LIN {X 0,Y 488.702,Z 333.231,A -85,B 0,C 180,E1 -6449.779,E2 -6449.779} C_VEL
LIN {X 0,Y 488.684,Z 333.228,A -85,B 0,C 180,E1 -6453.077,E2 -6453.077} C_VEL
LIN {X 0,Y 488.654,Z 333.238,A -85,B 0,C 180,E1 -6456.252,E2 -6456.252} C_VEL
LIN {X 0,Y 488.732,Z 333.224,A -85,B 0,C 180,E1 -6459.175,E2 -6459.175} C_VEL
LIN {X 0,Y 488.733,Z 333.22,A -85,B 0,C 180,E1 -6461.632,E2 -6461.632} C_VEL
LIN {X 0,Y 488.736,Z 333.23,A -85,B 0,C 180,E1 -6464.999,E2 -6464.999} C_VEL
LIN {X 0,Y 488.788,Z 333.224,A -85,B 0,C 180,E1 -6468.387,E2 -6468.387} C_VEL
LIN {X 0,Y 488.762,Z 333.222,A -85,B 0,C 180,E1 -6471.733,E2 -6471.733} C_VEL
LIN {X 0,Y 488.788,Z 333.223,A -85,B 0,C 180,E1 -6474.223,E2 -6474.223} C_VEL
LIN {X 0,Y 488.932,Z 333.202,A -85,B 0,C 180,E1 -6477.528,E2 -6477.528} C_VEL
LIN {X 0,Y 488.896,Z 333.211,A -85,B 0,C 180,E1 -6480.824,E2 -6480.824} C_VEL
LIN {X 0,Y 488.93,Z 333.21,A -85,B 0,C 180,E1 -6482.471,E2 -6482.471} C_VEL
LIN {X 0,Y 488.81,Z 333.217,A -85,B 0,C 180,E1 -6485.776,E2 -6485.776} C_VEL
LIN {X 0,Y 488.742,Z 333.23,A -85,B 0,C 180,E1 -6488.268,E2 -6488.268} C_VEL
LIN {X 0,Y 488.767,Z 333.222,A -85,B 0,C 180,E1 -6491.613,E2 -6491.613} C_VEL
LIN {X 0,Y 488.744,Z 333.227,A -85,B 0,C 180,E1 -6495.001,E2 -6495.001} C_VEL
LIN {X 0,Y 488.729,Z 333.235,A -85,B 0,C 180,E1 -6498.443,E2 -6498.443} C_VEL
LIN {X 0,Y 488.692,Z 333.227,A -85,B 0,C 180,E1 -6501.071,E2 -6501.071} C_VEL
LIN {X 0,Y 488.654,Z 333.233,A -85,B 0,C 180,E1 -6503.747,E2 -6503.747} C_VEL
LIN {X 0,Y 488.683,Z 333.233,A -85,B 0,C 180,E1 -6506.922,E2 -6506.922} C_VEL
LIN {X 0,Y 488.701,Z 333.232,A -85,B 0,C 180,E1 -6510.221,E2 -6510.221} C_VEL
LIN {X 0,Y 488.696,Z 333.23,A -85,B 0,C 180,E1 -6513.481,E2 -6513.481} C_VEL
LIN {X 0,Y 488.635,Z 333.246,A -85,B 0,C 180,E1 -6516.35,E2 -6516.35} C_VEL
LIN {X 0,Y 488.661,Z 333.236,A -85,B 0,C 180,E1 -6519.258,E2 -6519.258} C_VEL
LIN {X 0,Y 488.636,Z 333.244,A -85,B 0,C 180,E1 -6522.532,E2 -6522.532} C_VEL
LIN {X 0,Y 488.684,Z 333.234,A -85,B 0,C 180,E1 -6525.198,E2 -6525.198} C_VEL
LIN {X 0,Y 488.632,Z 333.245,A -85,B 0,C 180,E1 -6528.579,E2 -6528.579} C_VEL
LIN {X 0,Y 488.64,Z 333.243,A -85,B 0,C 180,E1 -6531.798,E2 -6531.798} C_VEL
LIN {X 0,Y 488.704,Z 333.232,A -85,B 0,C 180,E1 -6535.056,E2 -6535.056} C_VEL
LIN {X 0,Y 488.685,Z 333.24,A -85,B 0,C 180,E1 -6538.05,E2 -6538.05} C_VEL
LIN {X 0,Y 488.692,Z 333.232,A -85,B 0,C 180,E1 -6540.729,E2 -6540.729} C_VEL
LIN {X 0,Y 488.709,Z 333.391,A -85,B 0,C 180,E1 -6543.9,E2 -6543.9} C_VEL
LIN {X 0,Y 491.166,Z 344.956,A -85,B 0,C 180,E1 -6545.98,E2 -6545.98} C_VEL
LIN {X 0,Y 491.203,Z 350.07,A -85,B 0,C 180,E1 -6546.832,E2 -6546.832} C_VEL
LIN {X 0,Y 490.392,Z 368.886,A -85,B 0,C 180,E1 -6549.884,E2 -6549.884} C_VEL
LIN {X 0,Y 490.314,Z 371.302,A -85,B 0,C 180,E1 -6550.273,E2 -6550.273} C_VEL
LIN {X 0,Y 493.534,Z 389.01,A -85,B 0,C 180,E1 -6550.687,E2 -6550.687} C_VEL
LIN {X 0,Y 492.513,Z 509.403,A -85,B 0,C 180,E1 -6552.484,E2 -6552.484} C_VEL
LIN {X 0,Y 492.126,Z 523.948,A -85,B 0,C 180,E1 -6552.874,E2 -6552.874} C_VEL
LIN {X 0,Y 491.704,Z 538.324,A -85,B 0,C 180,E1 -6553.444,E2 -6553.444} C_VEL
LIN {X 0,Y 491.255,Z 551.142,A -85,B 0,C 180,E1 -6554.123,E2 -6554.123} C_VEL
LIN {X 0,Y 490.687,Z 563.612,A -85,B 0,C 180,E1 -6554.955,E2 -6554.955} C_VEL
LIN {X 0,Y 490.137,Z 575.001,A -85,B 0,C 180,E1 -6555.893,E2 -6555.893} C_VEL
LIN {X 0,Y 489.549,Z 585.47,A -85,B 0,C 180,E1 -6556.933,E2 -6556.933} C_VEL
LIN {X 0,Y 489.174,Z 596.158,A -85,B 0,C 180,E1 -6558.224,E2 -6558.224} C_VEL
LIN {X 0,Y 488.668,Z 605.74,A -85,B 0,C 180,E1 -6559.645,E2 -6559.645} C_VEL
LIN {X 0,Y 488.349,Z 613.708,A -85,B 0,C 180,E1 -6561.102,E2 -6561.102} C_VEL
LIN {X 0,Y 488.106,Z 620.121,A -85,B 0,C 180,E1 -6562.556,E2 -6562.556} C_VEL
LIN {X 0,Y 488.051,Z 625.81,A -85,B 0,C 180,E1 -6564.216,E2 -6564.216} C_VEL
LIN {X 0,Y 487.909,Z 629.938,A -85,B 0,C 180,E1 -6565.871,E2 -6565.871} C_VEL
LIN {X 0,Y 487.955,Z 631.458,A -85,B 0,C 180,E1 -6566.699,E2 -6566.699} C_VEL
LIN {X 0,Y 487.885,Z 633.463,A -85,B 0,C 180,E1 -6568.35,E2 -6568.35} C_VEL
LIN {X 0,Y 487.817,Z 634.126,A -85,B 0,C 180,E1 -6570.001,E2 -6570.001} C_VEL
LIN {X 0,Y 487.886,Z 633.459,A -85,B 0,C 180,E1 -6571.652,E2 -6571.652} C_VEL
LIN {X 0,Y 487.956,Z 631.449,A -85,B 0,C 180,E1 -6573.304,E2 -6573.304} C_VEL
LIN {X 0,Y 487.962,Z 628.05,A -85,B 0,C 180,E1 -6574.959,E2 -6574.959} C_VEL
LIN {X 0,Y 488.042,Z 623.66,A -85,B 0,C 180,E1 -6576.472,E2 -6576.472} C_VEL
LIN {X 0,Y 488.17,Z 618.444,A -85,B 0,C 180,E1 -6577.862,E2 -6577.862} C_VEL
LIN {X 0,Y 488.422,Z 611.598,A -85,B 0,C 180,E1 -6579.317,E2 -6579.317} C_VEL
LIN {X 0,Y 488.818,Z 603.102,A -85,B 0,C 180,E1 -6580.774,E2 -6580.774} C_VEL
LIN {X 0,Y 489.194,Z 594.847,A -85,B 0,C 180,E1 -6581.946,E2 -6581.946} C_VEL
LIN {X 0,Y 489.581,Z 585.447,A -85,B 0,C 180,E1 -6583.068,E2 -6583.068} C_VEL
LIN {X 0,Y 490.123,Z 574.974,A -85,B 0,C 180,E1 -6584.11,E2 -6584.11} C_VEL
LIN {X 0,Y 490.661,Z 563.574,A -85,B 0,C 180,E1 -6585.048,E2 -6585.048} C_VEL
LIN {X 0,Y 491.228,Z 551.097,A -85,B 0,C 180,E1 -6585.881,E2 -6585.881} C_VEL
LIN {X 0,Y 491.808,Z 537.148,A -85,B 0,C 180,E1 -6586.608,E2 -6586.608} C_VEL
LIN {X 0,Y 492.15,Z 523.043,A -85,B 0,C 180,E1 -6587.157,E2 -6587.157} C_VEL
LIN {X 0,Y 492.538,Z 509.287,A -85,B 0,C 180,E1 -6587.518,E2 -6587.518} C_VEL
LIN {X 0,Y 493.537,Z 388.937,A -85,B 0,C 180,E1 -6589.313,E2 -6589.313} C_VEL
LIN {X 0,Y 490.294,Z 371.281,A -85,B 0,C 180,E1 -6589.73,E2 -6589.73} C_VEL
LIN {X 0,Y 491.158,Z 351.392,A -85,B 0,C 180,E1 -6592.951,E2 -6592.951} C_VEL
LIN {X 0,Y 491.288,Z 346.01,A -85,B 0,C 180,E1 -6593.837,E2 -6593.837} C_VEL
LIN {X 0,Y 488.696,Z 333.239,A -85,B 0,C 180,E1 -6596.132,E2 -6596.132} C_VEL
LIN {X 0,Y 488.703,Z 333.237,A -85,B 0,C 180,E1 -6599.273,E2 -6599.273} C_VEL
LIN {X 0,Y 488.707,Z 333.233,A -85,B 0,C 180,E1 -6602.148,E2 -6602.148} C_VEL
LIN {X 0,Y 488.72,Z 333.234,A -85,B 0,C 180,E1 -6605.116,E2 -6605.116} C_VEL
LIN {X 0,Y 488.682,Z 333.234,A -85,B 0,C 180,E1 -6608.201,E2 -6608.201} C_VEL
LIN {X 0,Y 488.723,Z 333.229,A -85,B 0,C 180,E1 -6610.345,E2 -6610.345} C_VEL
LIN {X 0,Y 488.691,Z 333.234,A -85,B 0,C 180,E1 -6613.655,E2 -6613.655} C_VEL
LIN {X 0,Y 488.692,Z 333.237,A -85,B 0,C 180,E1 -6616.346,E2 -6616.346} C_VEL
LIN {X 0,Y 488.738,Z 333.228,A -85,B 0,C 180,E1 -6619.677,E2 -6619.677} C_VEL
LIN {X 0,Y 488.675,Z 333.238,A -85,B 0,C 180,E1 -6622.841,E2 -6622.841} C_VEL
LIN {X 0,Y 488.735,Z 333.231,A -85,B 0,C 180,E1 -6625.888,E2 -6625.888} C_VEL
LIN {X 0,Y 488.697,Z 333.236,A -85,B 0,C 180,E1 -6628.821,E2 -6628.821} C_VEL
LIN {X 0,Y 488.714,Z 333.239,A -85,B 0,C 180,E1 -6631.669,E2 -6631.669} C_VEL
LIN {X 0,Y 488.702,Z 333.235,A -85,B 0,C 180,E1 -6634.96,E2 -6634.96} C_VEL
LIN {X 0,Y 488.739,Z 333.298,A -85,B 0,C 180,E1 -6636.726,E2 -6636.726} C_VEL
LIN {X 0,Y 490.353,Z 342.584,A -85,B 0,C 180,E1 -6638.308,E2 -6638.308} C_VEL
LIN {X 0,Y 490.033,Z 361.132,A -85,B 0,C 180,E1 -6641.346,E2 -6641.346} C_VEL
LIN {X 0,Y 489.795,Z 376.155,A -85,B 0,C 180,E1 -6643.82,E2 -6643.82} C_VEL
LIN {X 0,Y 491.76,Z 387.528,A -85,B 0,C 180,E1 -6644.09,E2 -6644.09} C_VEL
LIN {X 0,Y 490.807,Z 484.773,A -85,B 0,C 180,E1 -6645.7,E2 -6645.7} C_VEL
LIN {X 0,Y 490.587,Z 497.505,A -85,B 0,C 180,E1 -6646.063,E2 -6646.063} C_VEL
LIN {X 0,Y 490.274,Z 509.826,A -85,B 0,C 180,E1 -6646.583,E2 -6646.583} C_VEL
LIN {X 0,Y 489.978,Z 521.787,A -85,B 0,C 180,E1 -6647.256,E2 -6647.256} C_VEL
LIN {X 0,Y 489.692,Z 533.257,A -85,B 0,C 180,E1 -6648.094,E2 -6648.094} C_VEL
LIN {X 0,Y 489.302,Z 543.523,A -85,B 0,C 180,E1 -6649.029,E2 -6649.029} C_VEL
LIN {X 0,Y 488.952,Z 552.812,A -85,B 0,C 180,E1 -6650.068,E2 -6650.068} C_VEL
LIN {X 0,Y 488.605,Z 561.725,A -85,B 0,C 180,E1 -6651.313,E2 -6651.313} C_VEL
LIN {X 0,Y 488.371,Z 568.89,A -85,B 0,C 180,E1 -6652.558,E2 -6652.558} C_VEL
LIN {X 0,Y 488.235,Z 575.028,A -85,B 0,C 180,E1 -6653.912,E2 -6653.912} C_VEL
LIN {X 0,Y 487.996,Z 579.059,A -85,B 0,C 180,E1 -6655.043,E2 -6655.043} C_VEL
LIN {X 0,Y 488.112,Z 581.377,A -85,B 0,C 180,E1 -6655.872,E2 -6655.872} C_VEL
LIN {X 0,Y 488.025,Z 583.275,A -85,B 0,C 180,E1 -6656.698,E2 -6656.698} C_VEL
LIN {X 0,Y 488,Z 584.743,A -85,B 0,C 180,E1 -6657.524,E2 -6657.524} C_VEL
LIN {X 0,Y 487.837,Z 586.379,A -85,B 0,C 180,E1 -6659.175,E2 -6659.175} C_VEL
LIN {X 0,Y 487.825,Z 586.609,A -85,B 0,C 180,E1 -6660,E2 -6660} C_VEL
LIN {X 0,Y 487.837,Z 586.402,A -85,B 0,C 180,E1 -6660.826,E2 -6660.826} C_VEL
LIN {X 0,Y 487.994,Z 584.776,A -85,B 0,C 180,E1 -6662.476,E2 -6662.476} C_VEL
LIN {X 0,Y 487.999,Z 583.356,A -85,B 0,C 180,E1 -6663.303,E2 -6663.303} C_VEL
LIN {X 0,Y 488.055,Z 580.39,A -85,B 0,C 180,E1 -6664.543,E2 -6664.543} C_VEL
LIN {X 0,Y 488.226,Z 575.193,A -85,B 0,C 180,E1 -6666.086,E2 -6666.086} C_VEL
LIN {X 0,Y 488.304,Z 569.158,A -85,B 0,C 180,E1 -6667.443,E2 -6667.443} C_VEL
LIN {X 0,Y 488.581,Z 562.093,A -85,B 0,C 180,E1 -6668.687,E2 -6668.687} C_VEL
LIN {X 0,Y 488.904,Z 553.302,A -85,B 0,C 180,E1 -6669.933,E2 -6669.933} C_VEL
LIN {X 0,Y 489.268,Z 544.258,A -85,B 0,C 180,E1 -6670.972,E2 -6670.972} C_VEL
LIN {X 0,Y 489.6,Z 534.233,A -85,B 0,C 180,E1 -6671.908,E2 -6671.908} C_VEL
LIN {X 0,Y 489.938,Z 522.917,A -85,B 0,C 180,E1 -6672.761,E2 -6672.761} C_VEL
LIN {X 0,Y 490.276,Z 510.773,A -85,B 0,C 180,E1 -6673.47,E2 -6673.47} C_VEL
LIN {X 0,Y 490.621,Z 497.552,A -85,B 0,C 180,E1 -6674.042,E2 -6674.042} C_VEL
LIN {X 0,Y 490.877,Z 485.355,A -85,B 0,C 180,E1 -6674.404,E2 -6674.404} C_VEL
LIN {X 0,Y 491.124,Z 459.02,A -85,B 0,C 180,E1 -6674.847,E2 -6674.847} C_VEL
LIN {X 0,Y 491.597,Z 386.183,A -85,B 0,C 180,E1 -6676.007,E2 -6676.007} C_VEL
LIN {X 0,Y 489.573,Z 374.944,A -85,B 0,C 180,E1 -6676.262,E2 -6676.262} C_VEL
LIN {X 0,Y 489.986,Z 357.352,A -85,B 0,C 180,E1 -6679.263,E2 -6679.263} C_VEL
LIN {X 0,Y 490.237,Z 342.024,A -85,B 0,C 180,E1 -6681.884,E2 -6681.884} C_VEL
LIN {X 0,Y 488.753,Z 333.23,A -85,B 0,C 180,E1 -6683.467,E2 -6683.467} C_VEL
LIN {X 0,Y 488.797,Z 333.221,A -85,B 0,C 180,E1 -6686.943,E2 -6686.943} C_VEL
LIN {X 0,Y 488.715,Z 333.233,A -85,B 0,C 180,E1 -6690.363,E2 -6690.363} C_VEL
LIN {X 0,Y 488.74,Z 333.228,A -85,B 0,C 180,E1 -6693.484,E2 -6693.484} C_VEL
LIN {X 0,Y 488.678,Z 333.238,A -85,B 0,C 180,E1 -6696.353,E2 -6696.353} C_VEL
LIN {X 0,Y 488.699,Z 333.232,A -85,B 0,C 180,E1 -6699.255,E2 -6699.255} C_VEL
LIN {X 0,Y 488.693,Z 333.233,A -85,B 0,C 180,E1 -6702.526,E2 -6702.526} C_VEL
LIN {X 0,Y 488.693,Z 333.234,A -85,B 0,C 180,E1 -6705.431,E2 -6705.431} C_VEL
LIN {X 0,Y 488.681,Z 333.234,A -85,B 0,C 180,E1 -6708.581,E2 -6708.581} C_VEL
LIN {X 0,Y 488.667,Z 333.236,A -85,B 0,C 180,E1 -6709.017,E2 -6709.017} C_VEL
LIN {X 0,Y 488.004,Z 333.325,A -85,B 0,C 180,E1 -6709.705,E2 -6709.705} C_VEL
LIN {X 0,Y 485.141,Z 333.677,A -85,B 0,C 180,E1 -6710.822,E2 -6710.822} C_VEL
LIN {X 0,Y 482.717,Z 333.983,A -85,B 0,C 180,E1 -6711.722,E2 -6711.722} C_VEL
LIN {X 0,Y 481.679,Z 334.108,A -85,B 0,C 180,E1 -6712.418,E2 -6712.418} C_VEL
LIN {X 0,Y 481.596,Z 334.118,A -85,B 0,C 180,E1 -6712.653,E2 -6712.653} C_VEL
LIN {X 0,Y 481.683,Z 334.11,A -85,B 0,C 180,E1 -6715.316,E2 -6715.316} C_VEL
LIN {X 0,Y 481.627,Z 334.115,A -85,B 0,C 180,E1 -6718.309,E2 -6718.309} C_VEL
LIN {X 0,Y 481.657,Z 334.117,A -85,B 0,C 180,E1 -6721.215,E2 -6721.215} C_VEL
LIN {X 0,Y 481.621,Z 334.119,A -85,B 0,C 180,E1 -6724.037,E2 -6724.037} C_VEL
LIN {X 0,Y 481.639,Z 334.155,A -85,B 0,C 180,E1 -6724.823,E2 -6724.823} C_VEL
LIN {X 0,Y 484.1,Z 346.337,A -85,B 0,C 180,E1 -6727.147,E2 -6727.147} C_VEL
LIN {X 0,Y 483.546,Z 360.333,A -85,B 0,C 180,E1 -6729.584,E2 -6729.584} C_VEL
LIN {X 0,Y 483.402,Z 362.996,A -85,B 0,C 180,E1 -6730.041,E2 -6730.041} C_VEL
LIN {X 0,Y 486.825,Z 379.799,A -85,B 0,C 180,E1 -6730.449,E2 -6730.449} C_VEL
LIN {X 0,Y 485.833,Z 498.193,A -85,B 0,C 180,E1 -6732.232,E2 -6732.232} C_VEL
LIN {X 0,Y 485.466,Z 512.773,A -85,B 0,C 180,E1 -6732.595,E2 -6732.595} C_VEL
LIN {X 0,Y 485.165,Z 526.114,A -85,B 0,C 180,E1 -6733.099,E2 -6733.099} C_VEL
LIN {X 0,Y 484.665,Z 537.87,A -85,B 0,C 180,E1 -6733.682,E2 -6733.682} C_VEL
LIN {X 0,Y 484.068,Z 551.218,A -85,B 0,C 180,E1 -6734.526,E2 -6734.526} C_VEL
LIN {X 0,Y 483.463,Z 563.197,A -85,B 0,C 180,E1 -6735.476,E2 -6735.476} C_VEL
LIN {X 0,Y 482.834,Z 574.12,A -85,B 0,C 180,E1 -6736.532,E2 -6736.532} C_VEL
LIN {X 0,Y 482.362,Z 584.598,A -85,B 0,C 180,E1 -6737.764,E2 -6737.764} C_VEL
LIN {X 0,Y 481.876,Z 593.784,A -85,B 0,C 180,E1 -6739.069,E2 -6739.069} C_VEL
LIN {X 0,Y 481.475,Z 602.295,A -85,B 0,C 180,E1 -6740.547,E2 -6740.547} C_VEL
LIN {X 0,Y 481.176,Z 609.155,A -85,B 0,C 180,E1 -6742.023,E2 -6742.023} C_VEL
LIN {X 0,Y 481.033,Z 614.484,A -85,B 0,C 180,E1 -6743.463,E2 -6743.463} C_VEL
LIN {X 0,Y 480.898,Z 618.792,A -85,B 0,C 180,E1 -6744.968,E2 -6744.968} C_VEL
LIN {X 0,Y 480.887,Z 622.208,A -85,B 0,C 180,E1 -6746.647,E2 -6746.647} C_VEL
LIN {X 0,Y 480.791,Z 624.243,A -85,B 0,C 180,E1 -6748.323,E2 -6748.323} C_VEL
LIN {X 0,Y 480.742,Z 624.947,A -85,B 0,C 180,E1 -6749.999,E2 -6749.999} C_VEL
LIN {X 0,Y 480.79,Z 624.327,A -85,B 0,C 180,E1 -6751.674,E2 -6751.674} C_VEL
LIN {X 0,Y 480.886,Z 622.372,A -85,B 0,C 180,E1 -6753.35,E2 -6753.35} C_VEL
LIN {X 0,Y 480.897,Z 619.029,A -85,B 0,C 180,E1 -6755.029,E2 -6755.029} C_VEL
LIN {X 0,Y 481.012,Z 614.202,A -85,B 0,C 180,E1 -6756.711,E2 -6756.711} C_VEL
LIN {X 0,Y 481.246,Z 607.745,A -85,B 0,C 180,E1 -6758.396,E2 -6758.396} C_VEL
LIN {X 0,Y 481.578,Z 600.556,A -85,B 0,C 180,E1 -6759.872,E2 -6759.872} C_VEL
LIN {X 0,Y 481.938,Z 593.021,A -85,B 0,C 180,E1 -6761.139,E2 -6761.139} C_VEL
LIN {X 0,Y 482.299,Z 584.534,A -85,B 0,C 180,E1 -6762.337,E2 -6762.337} C_VEL
LIN {X 0,Y 482.82,Z 574.963,A -85,B 0,C 180,E1 -6763.466,E2 -6763.466} C_VEL
LIN {X 0,Y 483.398,Z 564.21,A -85,B 0,C 180,E1 -6764.523,E2 -6764.523} C_VEL
LIN {X 0,Y 484.013,Z 552.449,A -85,B 0,C 180,E1 -6765.473,E2 -6765.473} C_VEL
LIN {X 0,Y 484.521,Z 541.228,A -85,B 0,C 180,E1 -6766.212,E2 -6766.212} C_VEL
LIN {X 0,Y 485.086,Z 528.046,A -85,B 0,C 180,E1 -6766.901,E2 -6766.901} C_VEL
LIN {X 0,Y 485.484,Z 513.858,A -85,B 0,C 180,E1 -6767.457,E2 -6767.457} C_VEL
LIN {X 0,Y 485.818,Z 500.184,A -85,B 0,C 180,E1 -6767.82,E2 -6767.82} C_VEL
LIN {X 0,Y 486.905,Z 380.439,A -85,B 0,C 180,E1 -6769.629,E2 -6769.629} C_VEL
LIN {X 0,Y 483.411,Z 362.985,A -85,B 0,C 180,E1 -6770.052,E2 -6770.052} C_VEL
LIN {X 0,Y 484.112,Z 346.87,A -85,B 0,C 180,E1 -6772.849,E2 -6772.849} C_VEL
LIN {X 0,Y 482.469,Z 337.99,A -85,B 0,C 180,E1 -6774.527,E2 -6774.527} C_VEL
LIN {X 0,Y 481.632,Z 334.12,A -85,B 0,C 180,E1 -6775.284,E2 -6775.284} C_VEL
LIN {X 0,Y 481.643,Z 334.115,A -85,B 0,C 180,E1 -6777.834,E2 -6777.834} C_VEL
LIN {X 0,Y 481.624,Z 334.121,A -85,B 0,C 180,E1 -6780.711,E2 -6780.711} C_VEL
LIN {X 0,Y 481.669,Z 334.111,A -85,B 0,C 180,E1 -6783.728,E2 -6783.728} C_VEL
LIN {X 0,Y 481.611,Z 334.121,A -85,B 0,C 180,E1 -6786.746,E2 -6786.746} C_VEL
LIN {X 0,Y 481.647,Z 334.11,A -85,B 0,C 180,E1 -6789.941,E2 -6789.941} C_VEL
LIN {X 0,Y 481.609,Z 334.118,A -85,B 0,C 180,E1 -6793.301,E2 -6793.301} C_VEL
LIN {X 0,Y 481.642,Z 334.111,A -85,B 0,C 180,E1 -6795.64,E2 -6795.64} C_VEL
LIN {X 0,Y 481.615,Z 334.121,A -85,B 0,C 180,E1 -6798.954,E2 -6798.954} C_VEL
LIN {X 0,Y 481.637,Z 334.106,A -85,B 0,C 180,E1 -6801.993,E2 -6801.993} C_VEL
LIN {X 0,Y 481.669,Z 334.108,A -85,B 0,C 180,E1 -6805.316,E2 -6805.316} C_VEL
LIN {X 0,Y 481.626,Z 334.109,A -85,B 0,C 180,E1 -6808.31,E2 -6808.31} C_VEL
LIN {X 0,Y 481.645,Z 334.111,A -85,B 0,C 180,E1 -6811.215,E2 -6811.215} C_VEL
LIN {X 0,Y 481.615,Z 334.105,A -85,B 0,C 180,E1 -6814.038,E2 -6814.038} C_VEL
LIN {X 0,Y 481.66,Z 334.115,A -85,B 0,C 180,E1 -6816.811,E2 -6816.811} C_VEL
LIN {X 0,Y 481.679,Z 334.1,A -85,B 0,C 180,E1 -6819.502,E2 -6819.502} C_VEL
LIN {X 0,Y 481.67,Z 334.101,A -85,B 0,C 180,E1 -6822.157,E2 -6822.157} C_VEL
LIN {X 0,Y 481.721,Z 334.107,A -85,B 0,C 180,E1 -6824.775,E2 -6824.775} C_VEL
LIN {X 0,Y 481.734,Z 334.101,A -85,B 0,C 180,E1 -6828.215,E2 -6828.215} C_VEL
LIN {X 0,Y 481.718,Z 334.099,A -85,B 0,C 180,E1 -6831.611,E2 -6831.611} C_VEL
LIN {X 0,Y 481.749,Z 334.099,A -85,B 0,C 180,E1 -6834.139,E2 -6834.139} C_VEL
LIN {X 0,Y 481.898,Z 334.078,A -85,B 0,C 180,E1 -6837.492,E2 -6837.492} C_VEL
LIN {X 0,Y 481.848,Z 334.089,A -85,B 0,C 180,E1 -6840.836,E2 -6840.836} C_VEL
LIN {X 0,Y 481.896,Z 334.087,A -85,B 0,C 180,E1 -6842.508,E2 -6842.508} C_VEL
LIN {X 0,Y 481.769,Z 334.095,A -85,B 0,C 180,E1 -6845.861,E2 -6845.861} C_VEL
LIN {X 0,Y 481.7,Z 334.108,A -85,B 0,C 180,E1 -6848.389,E2 -6848.389} C_VEL
LIN {X 0,Y 481.718,Z 334.101,A -85,B 0,C 180,E1 -6851.786,E2 -6851.786} C_VEL
LIN {X 0,Y 481.726,Z 334.1,A -85,B 0,C 180,E1 -6855.225,E2 -6855.225} C_VEL
LIN {X 0,Y 481.691,Z 334.108,A -85,B 0,C 180,E1 -6858.723,E2 -6858.723} C_VEL
LIN {X 0,Y 481.63,Z 334.105,A -85,B 0,C 180,E1 -6861.395,E2 -6861.395} C_VEL
LIN {X 0,Y 481.632,Z 334.111,A -85,B 0,C 180,E1 -6864.115,E2 -6864.115} C_VEL
LIN {X 0,Y 481.638,Z 334.109,A -85,B 0,C 180,E1 -6867.118,E2 -6867.118} C_VEL
LIN {X 0,Y 481.652,Z 334.104,A -85,B 0,C 180,E1 -6869.743,E2 -6869.743} C_VEL
LIN {X 0,Y 481.637,Z 334.113,A -85,B 0,C 180,E1 -6872.677,E2 -6872.677} C_VEL
LIN {X 0,Y 481.635,Z 334.111,A -85,B 0,C 180,E1 -6875.203,E2 -6875.203} C_VEL
LIN {X 0,Y 481.616,Z 334.119,A -85,B 0,C 180,E1 -6878.004,E2 -6878.004} C_VEL
LIN {X 0,Y 481.592,Z 334.117,A -85,B 0,C 180,E1 -6881.048,E2 -6881.048} C_VEL
LIN {X 0,Y 481.639,Z 334.117,A -85,B 0,C 180,E1 -6884.46,E2 -6884.46} C_VEL
LIN {X 0,Y 481.6,Z 334.118,A -85,B 0,C 180,E1 -6886.857,E2 -6886.857} C_VEL
LIN {X 0,Y 481.618,Z 334.121,A -85,B 0,C 180,E1 -6890.056,E2 -6890.056} C_VEL
LIN {X 0,Y 481.595,Z 334.118,A -85,B 0,C 180,E1 -6893.252,E2 -6893.252} C_VEL
LIN {X 0,Y 481.663,Z 334.115,A -85,B 0,C 180,E1 -6896.328,E2 -6896.328} C_VEL
LIN {X 0,Y 481.634,Z 334.113,A -85,B 0,C 180,E1 -6899.421,E2 -6899.421} C_VEL
LIN {X 0,Y 481.639,Z 334.117,A -85,B 0,C 180,E1 -6902.166,E2 -6902.166} C_VEL
LIN {X 0,Y 481.655,Z 334.175,A -85,B 0,C 180,E1 -6903.634,E2 -6903.634} C_VEL
LIN {X 0,Y 484.173,Z 345.973,A -85,B 0,C 180,E1 -6905.793,E2 -6905.793} C_VEL
LIN {X 0,Y 484.373,Z 350.071,A -85,B 0,C 180,E1 -6906.495,E2 -6906.495} C_VEL
LIN {X 0,Y 483.463,Z 370.03,A -85,B 0,C 180,E1 -6909.782,E2 -6909.782} C_VEL
LIN {X 0,Y 483.376,Z 371.316,A -85,B 0,C 180,E1 -6909.991,E2 -6909.991} C_VEL
LIN {X 0,Y 486.847,Z 390.105,A -85,B 0,C 180,E1 -6910.429,E2 -6910.429} C_VEL
LIN {X 0,Y 485.763,Z 509.343,A -85,B 0,C 180,E1 -6912.232,E2 -6912.232} C_VEL
LIN {X 0,Y 485.346,Z 523.819,A -85,B 0,C 180,E1 -6912.625,E2 -6912.625} C_VEL
LIN {X 0,Y 484.884,Z 538.339,A -85,B 0,C 180,E1 -6913.209,E2 -6913.209} C_VEL
LIN {X 0,Y 484.413,Z 551.103,A -85,B 0,C 180,E1 -6913.894,E2 -6913.894} C_VEL
LIN {X 0,Y 483.801,Z 563.547,A -85,B 0,C 180,E1 -6914.736,E2 -6914.736} C_VEL
LIN {X 0,Y 483.231,Z 574.935,A -85,B 0,C 180,E1 -6915.687,E2 -6915.687} C_VEL
LIN {X 0,Y 482.603,Z 585.404,A -85,B 0,C 180,E1 -6916.742,E2 -6916.742} C_VEL
LIN {X 0,Y 482.18,Z 595.054,A -85,B 0,C 180,E1 -6917.914,E2 -6917.914} C_VEL
LIN {X 0,Y 481.718,Z 604.407,A -85,B 0,C 180,E1 -6919.281,E2 -6919.281} C_VEL
LIN {X 0,Y 481.327,Z 612.632,A -85,B 0,C 180,E1 -6920.759,E2 -6920.759} C_VEL
LIN {X 0,Y 481.118,Z 618.386,A -85,B 0,C 180,E1 -6922.025,E2 -6922.025} C_VEL
LIN {X 0,Y 480.971,Z 623.909,A -85,B 0,C 180,E1 -6923.527,E2 -6923.527} C_VEL
LIN {X 0,Y 480.896,Z 627.993,A -85,B 0,C 180,E1 -6924.971,E2 -6924.971} C_VEL
LIN {X 0,Y 480.861,Z 631.39,A -85,B 0,C 180,E1 -6926.65,E2 -6926.65} C_VEL
LIN {X 0,Y 480.786,Z 633.396,A -85,B 0,C 180,E1 -6928.326,E2 -6928.326} C_VEL
LIN {X 0,Y 480.741,Z 634.059,A -85,B 0,C 180,E1 -6930.001,E2 -6930.001} C_VEL
LIN {X 0,Y 480.787,Z 633.392,A -85,B 0,C 180,E1 -6931.677,E2 -6931.677} C_VEL
LIN {X 0,Y 480.861,Z 631.382,A -85,B 0,C 180,E1 -6933.353,E2 -6933.353} C_VEL
LIN {X 0,Y 480.897,Z 627.983,A -85,B 0,C 180,E1 -6935.032,E2 -6935.032} C_VEL
LIN {X 0,Y 480.963,Z 623.095,A -85,B 0,C 180,E1 -6936.714,E2 -6936.714} C_VEL
LIN {X 0,Y 481.204,Z 616.563,A -85,B 0,C 180,E1 -6938.399,E2 -6938.399} C_VEL
LIN {X 0,Y 481.469,Z 609.294,A -85,B 0,C 180,E1 -6939.877,E2 -6939.877} C_VEL
LIN {X 0,Y 481.948,Z 600.295,A -85,B 0,C 180,E1 -6941.355,E2 -6941.355} C_VEL
LIN {X 0,Y 482.365,Z 590.845,A -85,B 0,C 180,E1 -6942.625,E2 -6942.625} C_VEL
LIN {X 0,Y 482.91,Z 580.387,A -85,B 0,C 180,E1 -6943.788,E2 -6943.788} C_VEL
LIN {X 0,Y 483.54,Z 568.842,A -85,B 0,C 180,E1 -6944.844,E2 -6944.844} C_VEL
LIN {X 0,Y 484.177,Z 556.033,A -85,B 0,C 180,E1 -6945.794,E2 -6945.794} C_VEL
LIN {X 0,Y 484.739,Z 543.534,A -85,B 0,C 180,E1 -6946.532,E2 -6946.532} C_VEL
LIN {X 0,Y 485.16,Z 530.397,A -85,B 0,C 180,E1 -6947.135,E2 -6947.135} C_VEL
LIN {X 0,Y 485.596,Z 517.164,A -85,B 0,C 180,E1 -6947.575,E2 -6947.575} C_VEL
LIN {X 0,Y 485.852,Z 503.427,A -85,B 0,C 180,E1 -6947.876,E2 -6947.876} C_VEL
LIN {X 0,Y 486.754,Z 389.035,A -85,B 0,C 180,E1 -6949.591,E2 -6949.591} C_VEL
LIN {X 0,Y 483.385,Z 371.212,A -85,B 0,C 180,E1 -6950.024,E2 -6950.024} C_VEL
LIN {X 0,Y 484.317,Z 351.368,A -85,B 0,C 180,E1 -6953.287,E2 -6953.287} C_VEL
LIN {X 0,Y 484.388,Z 347.292,A -85,B 0,C 180,E1 -6953.971,E2 -6953.971} C_VEL
LIN {X 0,Y 481.663,Z 334.115,A -85,B 0,C 180,E1 -6956.397,E2 -6956.397} C_VEL
LIN {X 0,Y 481.669,Z 334.113,A -85,B 0,C 180,E1 -6959.743,E2 -6959.743} C_VEL
LIN {X 0,Y 481.676,Z 334.109,A -85,B 0,C 180,E1 -6962.675,E2 -6962.675} C_VEL
LIN {X 0,Y 481.665,Z 334.113,A -85,B 0,C 180,E1 -6965.205,E2 -6965.205} C_VEL
LIN {X 0,Y 481.675,Z 334.11,A -85,B 0,C 180,E1 -6968.86,E2 -6968.86} C_VEL
LIN {X 0,Y 481.657,Z 334.109,A -85,B 0,C 180,E1 -6971.913,E2 -6971.913} C_VEL
LIN {X 0,Y 481.665,Z 334.111,A -85,B 0,C 180,E1 -6974.458,E2 -6974.458} C_VEL
LIN {X 0,Y 481.653,Z 334.111,A -85,B 0,C 180,E1 -6977.84,E2 -6977.84} C_VEL
LIN {X 0,Y 481.685,Z 334.112,A -85,B 0,C 180,E1 -6980.652,E2 -6980.652} C_VEL
LIN {X 0,Y 481.626,Z 334.113,A -85,B 0,C 180,E1 -6983.378,E2 -6983.378} C_VEL
LIN {X 0,Y 481.715,Z 334.108,A -85,B 0,C 180,E1 -6986.33,E2 -6986.33} C_VEL
LIN {X 0,Y 481.655,Z 334.113,A -85,B 0,C 180,E1 -6989.418,E2 -6989.418} C_VEL
LIN {X 0,Y 481.665,Z 334.118,A -85,B 0,C 180,E1 -6992.166,E2 -6992.166} C_VEL
LIN {X 0,Y 481.677,Z 334.111,A -85,B 0,C 180,E1 -6994.968,E2 -6994.968} C_VEL
LIN {X 0,Y 481.689,Z 334.227,A -85,B 0,C 180,E1 -6996.502,E2 -6996.502} C_VEL
LIN {X 0,Y 483.353,Z 342.916,A -85,B 0,C 180,E1 -6998.006,E2 -6998.006} C_VEL
LIN {X 0,Y 483.196,Z 358.881,A -85,B 0,C 180,E1 -7000.637,E2 -7000.637} C_VEL
LIN {X 0,Y 482.875,Z 376.63,A -85,B 0,C 180,E1 -7003.56,E2 -7003.56} C_VEL
LIN {X 0,Y 484.987,Z 388.328,A -85,B 0,C 180,E1 -7003.855,E2 -7003.855} C_VEL
LIN {X 0,Y 483.915,Z 485.736,A -85,B 0,C 180,E1 -7005.518,E2 -7005.518} C_VEL
LIN {X 0,Y 483.668,Z 498.857,A -85,B 0,C 180,E1 -7005.913,E2 -7005.913} C_VEL
LIN {X 0,Y 483.343,Z 511.96,A -85,B 0,C 180,E1 -7006.494,E2 -7006.494} C_VEL
LIN {X 0,Y 483.01,Z 522.847,A -85,B 0,C 180,E1 -7007.133,E2 -7007.133} C_VEL
LIN {X 0,Y 482.71,Z 534.656,A -85,B 0,C 180,E1 -7008.026,E2 -7008.026} C_VEL
LIN {X 0,Y 482.287,Z 544.752,A -85,B 0,C 180,E1 -7008.974,E2 -7008.974} C_VEL
LIN {X 0,Y 481.973,Z 553.029,A -85,B 0,C 180,E1 -7009.923,E2 -7009.923} C_VEL
LIN {X 0,Y 481.593,Z 561.972,A -85,B 0,C 180,E1 -7011.186,E2 -7011.186} C_VEL
LIN {X 0,Y 481.344,Z 569.154,A -85,B 0,C 180,E1 -7012.449,E2 -7012.449} C_VEL
LIN {X 0,Y 481.183,Z 575.48,A -85,B 0,C 180,E1 -7013.865,E2 -7013.865} C_VEL
LIN {X 0,Y 480.997,Z 580.582,A -85,B 0,C 180,E1 -7015.391,E2 -7015.391} C_VEL
LIN {X 0,Y 480.954,Z 583.595,A -85,B 0,C 180,E1 -7016.649,E2 -7016.649} C_VEL
LIN {X 0,Y 480.922,Z 585.068,A -85,B 0,C 180,E1 -7017.487,E2 -7017.487} C_VEL
LIN {X 0,Y 480.763,Z 586.704,A -85,B 0,C 180,E1 -7019.162,E2 -7019.162} C_VEL
LIN {X 0,Y 480.749,Z 586.932,A -85,B 0,C 180,E1 -7020,E2 -7020} C_VEL
LIN {X 0,Y 480.763,Z 586.719,A -85,B 0,C 180,E1 -7020.838,E2 -7020.838} C_VEL
LIN {X 0,Y 480.902,Z 585.08,A -85,B 0,C 180,E1 -7022.513,E2 -7022.513} C_VEL
LIN {X 0,Y 480.93,Z 583.646,A -85,B 0,C 180,E1 -7023.351,E2 -7023.351} C_VEL
LIN {X 0,Y 480.974,Z 580.659,A -85,B 0,C 180,E1 -7024.61,E2 -7024.61} C_VEL
LIN {X 0,Y 481.175,Z 575.598,A -85,B 0,C 180,E1 -7026.132,E2 -7026.132} C_VEL
LIN {X 0,Y 481.271,Z 569.358,A -85,B 0,C 180,E1 -7027.552,E2 -7027.552} C_VEL
LIN {X 0,Y 481.551,Z 562.249,A -85,B 0,C 180,E1 -7028.815,E2 -7028.815} C_VEL
LIN {X 0,Y 481.886,Z 553.41,A -85,B 0,C 180,E1 -7030.079,E2 -7030.079} C_VEL
LIN {X 0,Y 482.276,Z 544.294,A -85,B 0,C 180,E1 -7031.133,E2 -7031.133} C_VEL
LIN {X 0,Y 482.708,Z 532.954,A -85,B 0,C 180,E1 -7032.188,E2 -7032.188} C_VEL
LIN {X 0,Y 483.009,Z 522.158,A -85,B 0,C 180,E1 -7032.991,E2 -7032.991} C_VEL
LIN {X 0,Y 483.405,Z 509.451,A -85,B 0,C 180,E1 -7033.719,E2 -7033.719} C_VEL
LIN {X 0,Y 483.729,Z 496.374,A -85,B 0,C 180,E1 -7034.273,E2 -7034.273} C_VEL
LIN {X 0,Y 484.034,Z 483.21,A -85,B 0,C 180,E1 -7034.639,E2 -7034.639} C_VEL
LIN {X 0,Y 484.806,Z 387.332,A -85,B 0,C 180,E1 -7036.209,E2 -7036.209} C_VEL
LIN {X 0,Y 482.61,Z 375.126,A -85,B 0,C 180,E1 -7036.499,E2 -7036.499} C_VEL
LIN {X 0,Y 483.037,Z 357.359,A -85,B 0,C 180,E1 -7039.551,E2 -7039.551} C_VEL
LIN {X 0,Y 483.332,Z 344.404,A -85,B 0,C 180,E1 -7041.775,E2 -7041.775} C_VEL
LIN {X 0,Y 482.666,Z 339.253,A -85,B 0,C 180,E1 -7042.697,E2 -7042.697} C_VEL
LIN {X 0,Y 481.686,Z 334.112,A -85,B 0,C 180,E1 -7043.655,E2 -7043.655} C_VEL
LIN {X 0,Y 481.751,Z 334.099,A -85,B 0,C 180,E1 -7047.139,E2 -7047.139} C_VEL
LIN {X 0,Y 481.684,Z 334.109,A -85,B 0,C 180,E1 -7049.741,E2 -7049.741} C_VEL
LIN {X 0,Y 481.678,Z 334.107,A -85,B 0,C 180,E1 -7052.674,E2 -7052.674} C_VEL
LIN {X 0,Y 481.666,Z 334.108,A -85,B 0,C 180,E1 -7055.204,E2 -7055.204} C_VEL
LIN {X 0,Y 481.671,Z 334.107,A -85,B 0,C 180,E1 -7058.859,E2 -7058.859} C_VEL
LIN {X 0,Y 481.646,Z 334.114,A -85,B 0,C 180,E1 -7062.161,E2 -7062.161} C_VEL
LIN {X 0,Y 481.659,Z 334.115,A -85,B 0,C 180,E1 -7065.541,E2 -7065.541} C_VEL
LIN {X 0,Y 481.636,Z 334.113,A -85,B 0,C 180,E1 -7069.017,E2 -7069.017} C_VEL
LIN {X 0,Y 481.639,Z 334.115,A -85,B 0,C 180,E1 -7071.995,E2 -7071.995} C_VEL
LIN {X 0,Y 481.596,Z 334.118,A -85,B 0,C 180,E1 -7072.653,E2 -7072.653} C_VEL
LIN {X 0,Y 480.942,Z 334.204,A -85,B 0,C 180,E1 -7073.351,E2 -7073.351} C_VEL
LIN {X 0,Y 478.119,Z 334.554,A -85,B 0,C 180,E1 -7074.485,E2 -7074.485} C_VEL
LIN {X 0,Y 475.726,Z 334.852,A -85,B 0,C 180,E1 -7075.399,E2 -7075.399} C_VEL
LIN {X 0,Y 474.695,Z 334.979,A -85,B 0,C 180,E1 -7076.105,E2 -7076.105} C_VEL
LIN {X 0,Y 474.609,Z 334.989,A -85,B 0,C 180,E1 -7076.344,E2 -7076.344} C_VEL
LIN {X 0,Y 474.59,Z 334.995,A -85,B 0,C 180,E1 -7079.193,E2 -7079.193} C_VEL
LIN {X 0,Y 474.603,Z 334.993,A -85,B 0,C 180,E1 -7081.714,E2 -7081.714} C_VEL
LIN {X 0,Y 474.629,Z 335.103,A -85,B 0,C 180,E1 -7084.589,E2 -7084.589} C_VEL
LIN {X 0,Y 477.167,Z 347.672,A -85,B 0,C 180,E1 -7087.025,E2 -7087.025} C_VEL
LIN {X 0,Y 476.685,Z 360.401,A -85,B 0,C 180,E1 -7089.276,E2 -7089.276} C_VEL
LIN {X 0,Y 476.511,Z 363.066,A -85,B 0,C 180,E1 -7089.74,E2 -7089.74} C_VEL
LIN {X 0,Y 480.178,Z 381.305,A -85,B 0,C 180,E1 -7090.189,E2 -7090.189} C_VEL
LIN {X 0,Y 479.051,Z 499.75,A -85,B 0,C 180,E1 -7092,E2 -7092} C_VEL
LIN {X 0,Y 478.692,Z 513.85,A -85,B 0,C 180,E1 -7092.375,E2 -7092.375} C_VEL
LIN {X 0,Y 478.29,Z 527.421,A -85,B 0,C 180,E1 -7092.908,E2 -7092.908} C_VEL
LIN {X 0,Y 477.769,Z 539.787,A -85,B 0,C 180,E1 -7093.55,E2 -7093.55} C_VEL
LIN {X 0,Y 477.155,Z 552.715,A -85,B 0,C 180,E1 -7094.406,E2 -7094.406} C_VEL
LIN {X 0,Y 476.507,Z 564.442,A -85,B 0,C 180,E1 -7095.369,E2 -7095.369} C_VEL
LIN {X 0,Y 475.793,Z 576.139,A -85,B 0,C 180,E1 -7096.546,E2 -7096.546} C_VEL
LIN {X 0,Y 475.354,Z 585.932,A -85,B 0,C 180,E1 -7097.749,E2 -7097.749} C_VEL
LIN {X 0,Y 474.779,Z 595.206,A -85,B 0,C 180,E1 -7099.12,E2 -7099.12} C_VEL
LIN {X 0,Y 474.374,Z 603.468,A -85,B 0,C 180,E1 -7100.62,E2 -7100.62} C_VEL
LIN {X 0,Y 474.137,Z 609.225,A -85,B 0,C 180,E1 -7101.904,E2 -7101.904} C_VEL
LIN {X 0,Y 473.954,Z 614.899,A -85,B 0,C 180,E1 -7103.468,E2 -7103.468} C_VEL
LIN {X 0,Y 473.836,Z 618.861,A -85,B 0,C 180,E1 -7104.893,E2 -7104.893} C_VEL
LIN {X 0,Y 473.796,Z 622.276,A -85,B 0,C 180,E1 -7106.597,E2 -7106.597} C_VEL
LIN {X 0,Y 473.697,Z 624.311,A -85,B 0,C 180,E1 -7108.298,E2 -7108.298} C_VEL
LIN {X 0,Y 473.668,Z 625.014,A -85,B 0,C 180,E1 -7109.999,E2 -7109.999} C_VEL
LIN {X 0,Y 473.695,Z 624.394,A -85,B 0,C 180,E1 -7111.699,E2 -7111.699} C_VEL
LIN {X 0,Y 473.795,Z 622.438,A -85,B 0,C 180,E1 -7113.4,E2 -7113.4} C_VEL
LIN {X 0,Y 473.835,Z 619.095,A -85,B 0,C 180,E1 -7115.104,E2 -7115.104} C_VEL
LIN {X 0,Y 473.959,Z 614.267,A -85,B 0,C 180,E1 -7116.811,E2 -7116.811} C_VEL
LIN {X 0,Y 474.209,Z 607.81,A -85,B 0,C 180,E1 -7118.521,E2 -7118.521} C_VEL
LIN {X 0,Y 474.519,Z 600.621,A -85,B 0,C 180,E1 -7120.021,E2 -7120.021} C_VEL
LIN {X 0,Y 474.99,Z 591.727,A -85,B 0,C 180,E1 -7121.521,E2 -7121.521} C_VEL
LIN {X 0,Y 475.497,Z 582.385,A -85,B 0,C 180,E1 -7122.808,E2 -7122.808} C_VEL
LIN {X 0,Y 476.07,Z 572.036,A -85,B 0,C 180,E1 -7123.988,E2 -7123.988} C_VEL
LIN {X 0,Y 476.703,Z 560.621,A -85,B 0,C 180,E1 -7125.059,E2 -7125.059} C_VEL
LIN {X 0,Y 477.379,Z 547.97,A -85,B 0,C 180,E1 -7126.022,E2 -7126.022} C_VEL
LIN {X 0,Y 477.928,Z 535.995,A -85,B 0,C 180,E1 -7126.753,E2 -7126.753} C_VEL
LIN {X 0,Y 478.465,Z 522.035,A -85,B 0,C 180,E1 -7127.412,E2 -7127.412} C_VEL
LIN {X 0,Y 478.9,Z 507.863,A -85,B 0,C 180,E1 -7127.893,E2 -7127.893} C_VEL
LIN {X 0,Y 479.161,Z 494.362,A -85,B 0,C 180,E1 -7128.187,E2 -7128.187} C_VEL
LIN {X 0,Y 480.236,Z 381.552,A -85,B 0,C 180,E1 -7129.896,E2 -7129.896} C_VEL
LIN {X 0,Y 476.531,Z 363.026,A -85,B 0,C 180,E1 -7130.358,E2 -7130.358} C_VEL
LIN {X 0,Y 477.206,Z 348.2,A -85,B 0,C 180,E1 -7132.97,E2 -7132.97} C_VEL
LIN {X 0,Y 475.228,Z 338.047,A -85,B 0,C 180,E1 -7134.926,E2 -7134.926} C_VEL
LIN {X 0,Y 474.619,Z 334.992,A -85,B 0,C 180,E1 -7135.547,E2 -7135.547} C_VEL
LIN {X 0,Y 474.595,Z 334.993,A -85,B 0,C 180,E1 -7138.284,E2 -7138.284} C_VEL
LIN {X 0,Y 474.584,Z 334.999,A -85,B 0,C 180,E1 -7141.217,E2 -7141.217} C_VEL
LIN {X 0,Y 474.613,Z 334.99,A -85,B 0,C 180,E1 -7144.241,E2 -7144.241} C_VEL
LIN {X 0,Y 474.57,Z 334.995,A -85,B 0,C 180,E1 -7147.383,E2 -7147.383} C_VEL
LIN {X 0,Y 474.592,Z 334.99,A -85,B 0,C 180,E1 -7149.642,E2 -7149.642} C_VEL
LIN {X 0,Y 474.559,Z 334.999,A -85,B 0,C 180,E1 -7152.938,E2 -7152.938} C_VEL
LIN {X 0,Y 474.592,Z 334.989,A -85,B 0,C 180,E1 -7155.893,E2 -7155.893} C_VEL
LIN {X 0,Y 474.59,Z 334.995,A -85,B 0,C 180,E1 -7159.043,E2 -7159.043} C_VEL
LIN {X 0,Y 474.594,Z 334.983,A -85,B 0,C 180,E1 -7161.704,E2 -7161.704} C_VEL
LIN {X 0,Y 474.607,Z 334.994,A -85,B 0,C 180,E1 -7164.724,E2 -7164.724} C_VEL
LIN {X 0,Y 474.612,Z 334.98,A -85,B 0,C 180,E1 -7167.786,E2 -7167.786} C_VEL
LIN {X 0,Y 474.585,Z 334.994,A -85,B 0,C 180,E1 -7170.889,E2 -7170.889} C_VEL
LIN {X 0,Y 474.568,Z 334.982,A -85,B 0,C 180,E1 -7173.623,E2 -7173.623} C_VEL
LIN {X 0,Y 474.62,Z 334.991,A -85,B 0,C 180,E1 -7176.641,E2 -7176.641} C_VEL
LIN {X 0,Y 474.636,Z 334.978,A -85,B 0,C 180,E1 -7180.089,E2 -7180.089} C_VEL
LIN {X 0,Y 474.613,Z 334.989,A -85,B 0,C 180,E1 -7182.773,E2 -7182.773} C_VEL
LIN {X 0,Y 474.618,Z 334.985,A -85,B 0,C 180,E1 -7185.42,E2 -7185.42} C_VEL
LIN {X 0,Y 474.688,Z 334.977,A -85,B 0,C 180,E1 -7188.037,E2 -7188.037} C_VEL
LIN {X 0,Y 474.691,Z 334.974,A -85,B 0,C 180,E1 -7191.486,E2 -7191.486} C_VEL
LIN {X 0,Y 474.712,Z 334.975,A -85,B 0,C 180,E1 -7194.051,E2 -7194.051} C_VEL
LIN {X 0,Y 474.864,Z 334.955,A -85,B 0,C 180,E1 -7197.455,E2 -7197.455} C_VEL
LIN {X 0,Y 474.801,Z 334.967,A -85,B 0,C 180,E1 -7200.848,E2 -7200.848} C_VEL
LIN {X 0,Y 474.861,Z 334.962,A -85,B 0,C 180,E1 -7202.545,E2 -7202.545} C_VEL
LIN {X 0,Y 474.73,Z 334.972,A -85,B 0,C 180,E1 -7205.948,E2 -7205.948} C_VEL
LIN {X 0,Y 474.649,Z 334.986,A -85,B 0,C 180,E1 -7208.515,E2 -7208.515} C_VEL
LIN {X 0,Y 474.676,Z 334.98,A -85,B 0,C 180,E1 -7211.963,E2 -7211.963} C_VEL
LIN {X 0,Y 474.684,Z 334.977,A -85,B 0,C 180,E1 -7215.456,E2 -7215.456} C_VEL
LIN {X 0,Y 474.645,Z 334.983,A -85,B 0,C 180,E1 -7219.011,E2 -7219.011} C_VEL
LIN {X 0,Y 474.573,Z 334.985,A -85,B 0,C 180,E1 -7221.73,E2 -7221.73} C_VEL
LIN {X 0,Y 474.61,Z 334.992,A -85,B 0,C 180,E1 -7224.496,E2 -7224.496} C_VEL
LIN {X 0,Y 474.585,Z 334.987,A -85,B 0,C 180,E1 -7227.327,E2 -7227.327} C_VEL
LIN {X 0,Y 474.581,Z 334.99,A -85,B 0,C 180,E1 -7230.232,E2 -7230.232} C_VEL
LIN {X 0,Y 474.601,Z 334.986,A -85,B 0,C 180,E1 -7233.223,E2 -7233.223} C_VEL
LIN {X 0,Y 474.557,Z 334.999,A -85,B 0,C 180,E1 -7236.326,E2 -7236.326} C_VEL
LIN {X 0,Y 474.588,Z 334.99,A -85,B 0,C 180,E1 -7239.551,E2 -7239.551} C_VEL
LIN {X 0,Y 474.554,Z 334.994,A -85,B 0,C 180,E1 -7242.941,E2 -7242.941} C_VEL
LIN {X 0,Y 474.586,Z 334.994,A -85,B 0,C 180,E1 -7245.895,E2 -7245.895} C_VEL
LIN {X 0,Y 474.57,Z 334.993,A -85,B 0,C 180,E1 -7249.049,E2 -7249.049} C_VEL
LIN {X 0,Y 474.576,Z 334.995,A -85,B 0,C 180,E1 -7251.709,E2 -7251.709} C_VEL
LIN {X 0,Y 474.601,Z 334.991,A -85,B 0,C 180,E1 -7254.726,E2 -7254.726} C_VEL
LIN {X 0,Y 474.613,Z 334.992,A -85,B 0,C 180,E1 -7257.788,E2 -7257.788} C_VEL
LIN {X 0,Y 474.59,Z 334.988,A -85,B 0,C 180,E1 -7260.892,E2 -7260.892} C_VEL
LIN {X 0,Y 474.63,Z 335.128,A -85,B 0,C 180,E1 -7263.391,E2 -7263.391} C_VEL
LIN {X 0,Y 477.445,Z 348.493,A -85,B 0,C 180,E1 -7265.873,E2 -7265.873} C_VEL
LIN {X 0,Y 477.158,Z 358.021,A -85,B 0,C 180,E1 -7267.485,E2 -7267.485} C_VEL
LIN {X 0,Y 476.509,Z 371.171,A -85,B 0,C 180,E1 -7269.677,E2 -7269.677} C_VEL
LIN {X 0,Y 480.148,Z 390.913,A -85,B 0,C 180,E1 -7270.158,E2 -7270.158} C_VEL
LIN {X 0,Y 479.01,Z 509.285,A -85,B 0,C 180,E1 -7271.973,E2 -7271.973} C_VEL
LIN {X 0,Y 478.592,Z 523.758,A -85,B 0,C 180,E1 -7272.372,E2 -7272.372} C_VEL
LIN {X 0,Y 478.093,Z 538.143,A -85,B 0,C 180,E1 -7272.956,E2 -7272.956} C_VEL
LIN {X 0,Y 477.58,Z 551.132,A -85,B 0,C 180,E1 -7273.663,E2 -7273.663} C_VEL
LIN {X 0,Y 476.907,Z 563.482,A -85,B 0,C 180,E1 -7274.51,E2 -7274.51} C_VEL
LIN {X 0,Y 476.258,Z 576.042,A -85,B 0,C 180,E1 -7275.582,E2 -7275.582} C_VEL
LIN {X 0,Y 475.565,Z 587.234,A -85,B 0,C 180,E1 -7276.76,E2 -7276.76} C_VEL
LIN {X 0,Y 475.094,Z 597.271,A -85,B 0,C 180,E1 -7278.049,E2 -7278.049} C_VEL
LIN {X 0,Y 474.615,Z 605.606,A -85,B 0,C 180,E1 -7279.335,E2 -7279.335} C_VEL
LIN {X 0,Y 474.253,Z 613.574,A -85,B 0,C 180,E1 -7280.835,E2 -7280.835} C_VEL
LIN {X 0,Y 473.972,Z 619.986,A -85,B 0,C 180,E1 -7282.332,E2 -7282.332} C_VEL
LIN {X 0,Y 473.859,Z 625.675,A -85,B 0,C 180,E1 -7284.042,E2 -7284.042} C_VEL
LIN {X 0,Y 473.723,Z 629.803,A -85,B 0,C 180,E1 -7285.747,E2 -7285.747} C_VEL
LIN {X 0,Y 473.719,Z 632.495,A -85,B 0,C 180,E1 -7287.45,E2 -7287.45} C_VEL
LIN {X 0,Y 473.685,Z 633.827,A -85,B 0,C 180,E1 -7289.151,E2 -7289.151} C_VEL
LIN {X 0,Y 473.686,Z 633.825,A -85,B 0,C 180,E1 -7290.851,E2 -7290.851} C_VEL
LIN {X 0,Y 473.72,Z 632.489,A -85,B 0,C 180,E1 -7292.552,E2 -7292.552} C_VEL
LIN {X 0,Y 473.723,Z 629.793,A -85,B 0,C 180,E1 -7294.255,E2 -7294.255} C_VEL
LIN {X 0,Y 473.862,Z 626.85,A -85,B 0,C 180,E1 -7295.533,E2 -7295.533} C_VEL
LIN {X 0,Y 473.923,Z 621.59,A -85,B 0,C 180,E1 -7297.243,E2 -7297.243} C_VEL
LIN {X 0,Y 474.132,Z 616.495,A -85,B 0,C 180,E1 -7298.525,E2 -7298.525} C_VEL
LIN {X 0,Y 474.434,Z 609.226,A -85,B 0,C 180,E1 -7300.025,E2 -7300.025} C_VEL
LIN {X 0,Y 474.957,Z 600.226,A -85,B 0,C 180,E1 -7301.524,E2 -7301.524} C_VEL
LIN {X 0,Y 475.395,Z 590.776,A -85,B 0,C 180,E1 -7302.813,E2 -7302.813} C_VEL
LIN {X 0,Y 475.972,Z 580.317,A -85,B 0,C 180,E1 -7303.993,E2 -7303.993} C_VEL
LIN {X 0,Y 476.64,Z 568.772,A -85,B 0,C 180,E1 -7305.064,E2 -7305.064} C_VEL
LIN {X 0,Y 477.326,Z 555.962,A -85,B 0,C 180,E1 -7306.027,E2 -7306.027} C_VEL
LIN {X 0,Y 477.904,Z 544.013,A -85,B 0,C 180,E1 -7306.745,E2 -7306.745} C_VEL
LIN {X 0,Y 478.381,Z 530.325,A -85,B 0,C 180,E1 -7307.386,E2 -7307.386} C_VEL
LIN {X 0,Y 478.83,Z 517.089,A -85,B 0,C 180,E1 -7307.832,E2 -7307.832} C_VEL
LIN {X 0,Y 479.088,Z 503.348,A -85,B 0,C 180,E1 -7308.137,E2 -7308.137} C_VEL
LIN {X 0,Y 480.16,Z 390.66,A -85,B 0,C 180,E1 -7309.844,E2 -7309.844} C_VEL
LIN {X 0,Y 476.496,Z 371.144,A -85,B 0,C 180,E1 -7310.326,E2 -7310.326} C_VEL
LIN {X 0,Y 477.482,Z 351.537,A -85,B 0,C 180,E1 -7313.601,E2 -7313.601} C_VEL
LIN {X 0,Y 477.207,Z 347.226,A -85,B 0,C 180,E1 -7314.355,E2 -7314.355} C_VEL
LIN {X 0,Y 474.621,Z 334.991,A -85,B 0,C 180,E1 -7316.671,E2 -7316.671} C_VEL
LIN {X 0,Y 474.603,Z 334.993,A -85,B 0,C 180,E1 -7319.254,E2 -7319.254} C_VEL
LIN {X 0,Y 474.619,Z 334.988,A -85,B 0,C 180,E1 -7322.431,E2 -7322.431} C_VEL
LIN {X 0,Y 474.616,Z 334.992,A -85,B 0,C 180,E1 -7325.469,E2 -7325.469} C_VEL
LIN {X 0,Y 474.615,Z 334.987,A -85,B 0,C 180,E1 -7328.458,E2 -7328.458} C_VEL
LIN {X 0,Y 474.625,Z 334.986,A -85,B 0,C 180,E1 -7331.786,E2 -7331.786} C_VEL
LIN {X 0,Y 474.626,Z 334.988,A -85,B 0,C 180,E1 -7335.298,E2 -7335.298} C_VEL
LIN {X 0,Y 474.625,Z 334.988,A -85,B 0,C 180,E1 -7338.215,E2 -7338.215} C_VEL
LIN {X 0,Y 474.649,Z 334.986,A -85,B 0,C 180,E1 -7340.455,E2 -7340.455} C_VEL
LIN {X 0,Y 474.589,Z 334.99,A -85,B 0,C 180,E1 -7343.676,E2 -7343.676} C_VEL
LIN {X 0,Y 474.648,Z 334.987,A -85,B 0,C 180,E1 -7346.78,E2 -7346.78} C_VEL
LIN {X 0,Y 474.608,Z 334.994,A -85,B 0,C 180,E1 -7349.77,E2 -7349.77} C_VEL
LIN {X 0,Y 474.642,Z 334.991,A -85,B 0,C 180,E1 -7352.676,E2 -7352.676} C_VEL
LIN {X 0,Y 474.625,Z 334.993,A -85,B 0,C 180,E1 -7355.971,E2 -7355.971} C_VEL
LIN {X 0,Y 474.65,Z 335.182,A -85,B 0,C 180,E1 -7356.262,E2 -7356.262} C_VEL
LIN {X 0,Y 476.499,Z 344.59,A -85,B 0,C 180,E1 -7357.908,E2 -7357.908} C_VEL
LIN {X 0,Y 476.322,Z 360.612,A -85,B 0,C 180,E1 -7360.575,E2 -7360.575} C_VEL
LIN {X 0,Y 475.973,Z 376.806,A -85,B 0,C 180,E1 -7363.28,E2 -7363.28} C_VEL
LIN {X 0,Y 478.224,Z 389.099,A -85,B 0,C 180,E1 -7363.605,E2 -7363.605} C_VEL
LIN {X 0,Y 477.052,Z 485.764,A -85,B 0,C 180,E1 -7365.305,E2 -7365.305} C_VEL
LIN {X 0,Y 476.793,Z 498.978,A -85,B 0,C 180,E1 -7365.706,E2 -7365.706} C_VEL
LIN {X 0,Y 476.441,Z 512.1,A -85,B 0,C 180,E1 -7366.294,E2 -7366.294} C_VEL
LIN {X 0,Y 476.093,Z 523.588,A -85,B 0,C 180,E1 -7366.98,E2 -7366.98} C_VEL
LIN {X 0,Y 475.774,Z 534.879,A -85,B 0,C 180,E1 -7367.849,E2 -7367.849} C_VEL
LIN {X 0,Y 475.324,Z 544.992,A -85,B 0,C 180,E1 -7368.81,E2 -7368.81} C_VEL
LIN {X 0,Y 474.998,Z 553.285,A -85,B 0,C 180,E1 -7369.773,E2 -7369.773} C_VEL
LIN {X 0,Y 474.656,Z 560.919,A -85,B 0,C 180,E1 -7370.841,E2 -7370.841} C_VEL
LIN {X 0,Y 474.33,Z 568.357,A -85,B 0,C 180,E1 -7372.123,E2 -7372.123} C_VEL
LIN {X 0,Y 474.131,Z 575.087,A -85,B 0,C 180,E1 -7373.588,E2 -7373.588} C_VEL
LIN {X 0,Y 473.869,Z 579.691,A -85,B 0,C 180,E1 -7374.895,E2 -7374.895} C_VEL
LIN {X 0,Y 473.968,Z 582.019,A -85,B 0,C 180,E1 -7375.748,E2 -7375.748} C_VEL
LIN {X 0,Y 473.885,Z 583.924,A -85,B 0,C 180,E1 -7376.599,E2 -7376.599} C_VEL
LIN {X 0,Y 473.834,Z 585.399,A -85,B 0,C 180,E1 -7377.45,E2 -7377.45} C_VEL
LIN {X 0,Y 473.762,Z 586.413,A -85,B 0,C 180,E1 -7378.3,E2 -7378.3} C_VEL
LIN {X 0,Y 473.675,Z 587.256,A -85,B 0,C 180,E1 -7380,E2 -7380} C_VEL
LIN {X 0,Y 473.691,Z 587.036,A -85,B 0,C 180,E1 -7380.85,E2 -7380.85} C_VEL
LIN {X 0,Y 473.761,Z 586.404,A -85,B 0,C 180,E1 -7381.7,E2 -7381.7} C_VEL
LIN {X 0,Y 473.815,Z 585.381,A -85,B 0,C 180,E1 -7382.55,E2 -7382.55} C_VEL
LIN {X 0,Y 473.863,Z 583.932,A -85,B 0,C 180,E1 -7383.401,E2 -7383.401} C_VEL
LIN {X 0,Y 473.88,Z 580.924,A -85,B 0,C 180,E1 -7384.679,E2 -7384.679} C_VEL
LIN {X 0,Y 474.094,Z 576.838,A -85,B 0,C 180,E1 -7385.956,E2 -7385.956} C_VEL
LIN {X 0,Y 474.195,Z 570.568,A -85,B 0,C 180,E1 -7387.451,E2 -7387.451} C_VEL
LIN {X 0,Y 474.471,Z 563.721,A -85,B 0,C 180,E1 -7388.733,E2 -7388.733} C_VEL
LIN {X 0,Y 474.803,Z 555.107,A -85,B 0,C 180,E1 -7390.016,E2 -7390.016} C_VEL
LIN {X 0,Y 475.172,Z 546.29,A -85,B 0,C 180,E1 -7391.086,E2 -7391.086} C_VEL
LIN {X 0,Y 475.578,Z 536.654,A -85,B 0,C 180,E1 -7392.046,E2 -7392.046} C_VEL
LIN {X 0,Y 475.936,Z 525.517,A -85,B 0,C 180,E1 -7392.938,E2 -7392.938} C_VEL
LIN {X 0,Y 476.35,Z 514.206,A -85,B 0,C 180,E1 -7393.654,E2 -7393.654} C_VEL
LIN {X 0,Y 476.689,Z 502.121,A -85,B 0,C 180,E1 -7394.243,E2 -7394.243} C_VEL
LIN {X 0,Y 476.992,Z 488.794,A -85,B 0,C 180,E1 -7394.697,E2 -7394.697} C_VEL
LIN {X 0,Y 477.175,Z 474.652,A -85,B 0,C 180,E1 -7394.991,E2 -7394.991} C_VEL
LIN {X 0,Y 477.901,Z 387.926,A -85,B 0,C 180,E1 -7396.432,E2 -7396.432} C_VEL
LIN {X 0,Y 475.658,Z 375.318,A -85,B 0,C 180,E1 -7396.742,E2 -7396.742} C_VEL
LIN {X 0,Y 476.079,Z 358.607,A -85,B 0,C 180,E1 -7399.625,E2 -7399.625} C_VEL
LIN {X 0,Y 476.399,Z 345.738,A -85,B 0,C 180,E1 -7401.847,E2 -7401.847} C_VEL
LIN {X 0,Y 475.665,Z 340.382,A -85,B 0,C 180,E1 -7402.815,E2 -7402.815} C_VEL
LIN {X 0,Y 474.647,Z 334.989,A -85,B 0,C 180,E1 -7403.825,E2 -7403.825} C_VEL
LIN {X 0,Y 474.659,Z 334.988,A -85,B 0,C 180,E1 -7406.372,E2 -7406.372} C_VEL
LIN {X 0,Y 474.625,Z 334.985,A -85,B 0,C 180,E1 -7409.252,E2 -7409.252} C_VEL
LIN {X 0,Y 474.621,Z 334.989,A -85,B 0,C 180,E1 -7412.43,E2 -7412.43} C_VEL
LIN {X 0,Y 474.617,Z 334.988,A -85,B 0,C 180,E1 -7415.468,E2 -7415.468} C_VEL
LIN {X 0,Y 474.613,Z 334.988,A -85,B 0,C 180,E1 -7418.457,E2 -7418.457} C_VEL
LIN {X 0,Y 474.614,Z 334.994,A -85,B 0,C 180,E1 -7421.786,E2 -7421.786} C_VEL
LIN {X 0,Y 474.621,Z 334.986,A -85,B 0,C 180,E1 -7424.702,E2 -7424.702} C_VEL
LIN {X 0,Y 474.593,Z 334.996,A -85,B 0,C 180,E1 -7427.768,E2 -7427.768} C_VEL
LIN {X 0,Y 474.623,Z 334.986,A -85,B 0,C 180,E1 -7430.451,E2 -7430.451} C_VEL
LIN {X 0,Y 474.585,Z 334.996,A -85,B 0,C 180,E1 -7433.675,E2 -7433.675} C_VEL
LIN {X 0,Y 474.609,Z 334.989,A -85,B 0,C 180,E1 -7436.344,E2 -7436.344} C_VEL
LIN {X 0,Y 473.93,Z 335.077,A -85,B 0,C 180,E1 -7437.052,E2 -7437.052} C_VEL
LIN {X 0,Y 471.051,Z 335.433,A -85,B 0,C 180,E1 -7438.202,E2 -7438.202} C_VEL
LIN {X 0,Y 468.63,Z 335.738,A -85,B 0,C 180,E1 -7439.129,E2 -7439.129} C_VEL
LIN {X 0,Y 467.605,Z 335.864,A -85,B 0,C 180,E1 -7439.846,E2 -7439.846} C_VEL
LIN {X 0,Y 467.53,Z 335.871,A -85,B 0,C 180,E1 -7440.088,E2 -7440.088} C_VEL
LIN {X 0,Y 467.528,Z 335.869,A -85,B 0,C 180,E1 -7443.193,E2 -7443.193} C_VEL
LIN {X 0,Y 467.571,Z 335.965,A -85,B 0,C 180,E1 -7444.328,E2 -7444.328} C_VEL
LIN {X 0,Y 470.246,Z 349.007,A -85,B 0,C 180,E1 -7446.9,E2 -7446.9} C_VEL
LIN {X 0,Y 469.929,Z 357.918,A -85,B 0,C 180,E1 -7448.505,E2 -7448.505} C_VEL
LIN {X 0,Y 469.686,Z 363.121,A -85,B 0,C 180,E1 -7449.429,E2 -7449.429} C_VEL
LIN {X 0,Y 473.437,Z 381.687,A -85,B 0,C 180,E1 -7449.899,E2 -7449.899} C_VEL
LIN {X 0,Y 472.395,Z 496.874,A -85,B 0,C 180,E1 -7451.681,E2 -7451.681} C_VEL
LIN {X 0,Y 472.031,Z 511.067,A -85,B 0,C 180,E1 -7452.026,E2 -7452.026} C_VEL
LIN {X 0,Y 471.601,Z 525.134,A -85,B 0,C 180,E1 -7452.548,E2 -7452.548} C_VEL
LIN {X 0,Y 471.04,Z 538.191,A -85,B 0,C 180,E1 -7453.206,E2 -7453.206} C_VEL
LIN {X 0,Y 470.379,Z 551.365,A -85,B 0,C 180,E1 -7454.064,E2 -7454.064} C_VEL
LIN {X 0,Y 469.66,Z 563.343,A -85,B 0,C 180,E1 -7455.04,E2 -7455.04} C_VEL
LIN {X 0,Y 468.977,Z 574.264,A -85,B 0,C 180,E1 -7456.126,E2 -7456.126} C_VEL
LIN {X 0,Y 468.405,Z 584.847,A -85,B 0,C 180,E1 -7457.408,E2 -7457.408} C_VEL
LIN {X 0,Y 467.881,Z 593.925,A -85,B 0,C 180,E1 -7458.738,E2 -7458.738} C_VEL
LIN {X 0,Y 467.418,Z 602.436,A -85,B 0,C 180,E1 -7460.26,E2 -7460.26} C_VEL
LIN {X 0,Y 467.086,Z 609.295,A -85,B 0,C 180,E1 -7461.781,E2 -7461.781} C_VEL
LIN {X 0,Y 466.864,Z 615.343,A -85,B 0,C 180,E1 -7463.486,E2 -7463.486} C_VEL
LIN {X 0,Y 466.773,Z 618.929,A -85,B 0,C 180,E1 -7464.816,E2 -7464.816} C_VEL
LIN {X 0,Y 466.693,Z 622.344,A -85,B 0,C 180,E1 -7466.545,E2 -7466.545} C_VEL
LIN {X 0,Y 466.606,Z 624.378,A -85,B 0,C 180,E1 -7468.272,E2 -7468.272} C_VEL
LIN {X 0,Y 466.598,Z 625.081,A -85,B 0,C 180,E1 -7469.999,E2 -7469.999} C_VEL
LIN {X 0,Y 466.605,Z 624.461,A -85,B 0,C 180,E1 -7471.725,E2 -7471.725} C_VEL
LIN {X 0,Y 466.691,Z 622.504,A -85,B 0,C 180,E1 -7473.452,E2 -7473.452} C_VEL
LIN {X 0,Y 466.772,Z 619.161,A -85,B 0,C 180,E1 -7475.182,E2 -7475.182} C_VEL
LIN {X 0,Y 466.9,Z 614.333,A -85,B 0,C 180,E1 -7476.915,E2 -7476.915} C_VEL
LIN {X 0,Y 467.143,Z 607.876,A -85,B 0,C 180,E1 -7478.651,E2 -7478.651} C_VEL
LIN {X 0,Y 467.482,Z 600.686,A -85,B 0,C 180,E1 -7480.173,E2 -7480.173} C_VEL
LIN {X 0,Y 468.007,Z 591.791,A -85,B 0,C 180,E1 -7481.695,E2 -7481.695} C_VEL
LIN {X 0,Y 468.532,Z 582.449,A -85,B 0,C 180,E1 -7483.001,E2 -7483.001} C_VEL
LIN {X 0,Y 469.144,Z 572.099,A -85,B 0,C 180,E1 -7484.198,E2 -7484.198} C_VEL
LIN {X 0,Y 469.816,Z 560.683,A -85,B 0,C 180,E1 -7485.285,E2 -7485.285} C_VEL
LIN {X 0,Y 470.557,Z 548.03,A -85,B 0,C 180,E1 -7486.261,E2 -7486.261} C_VEL
LIN {X 0,Y 471.189,Z 534.635,A -85,B 0,C 180,E1 -7487.08,E2 -7487.08} C_VEL
LIN {X 0,Y 471.761,Z 520.792,A -85,B 0,C 180,E1 -7487.724,E2 -7487.724} C_VEL
LIN {X 0,Y 472.173,Z 506.999,A -85,B 0,C 180,E1 -7488.185,E2 -7488.185} C_VEL
LIN {X 0,Y 472.458,Z 492.809,A -85,B 0,C 180,E1 -7488.482,E2 -7488.482} C_VEL
LIN {X 0,Y 473.556,Z 382.584,A -85,B 0,C 180,E1 -7490.173,E2 -7490.173} C_VEL
LIN {X 0,Y 469.708,Z 362.993,A -85,B 0,C 180,E1 -7490.685,E2 -7490.685} C_VEL
LIN {X 0,Y 470.283,Z 349.53,A -85,B 0,C 180,E1 -7493.095,E2 -7493.095} C_VEL
LIN {X 0,Y 468.096,Z 338.418,A -85,B 0,C 180,E1 -7495.274,E2 -7495.274} C_VEL
LIN {X 0,Y 467.567,Z 335.87,A -85,B 0,C 180,E1 -7495.799,E2 -7495.799} C_VEL
LIN {X 0,Y 467.535,Z 335.876,A -85,B 0,C 180,E1 -7498.751,E2 -7498.751} C_VEL
LIN {X 0,Y 467.554,Z 335.87,A -85,B 0,C 180,E1 -7501.74,E2 -7501.74} C_VEL
LIN {X 0,Y 467.55,Z 335.874,A -85,B 0,C 180,E1 -7504.832,E2 -7504.832} C_VEL
LIN {X 0,Y 467.547,Z 335.867,A -85,B 0,C 180,E1 -7508.044,E2 -7508.044} C_VEL
LIN {X 0,Y 467.551,Z 335.87,A -85,B 0,C 180,E1 -7511.273,E2 -7511.273} C_VEL
LIN {X 0,Y 467.555,Z 335.872,A -85,B 0,C 180,E1 -7514.946,E2 -7514.946} C_VEL
LIN {X 0,Y 467.515,Z 335.872,A -85,B 0,C 180,E1 -7517.44,E2 -7517.44} C_VEL
LIN {X 0,Y 467.552,Z 335.866,A -85,B 0,C 180,E1 -7520.047,E2 -7520.047} C_VEL
LIN {X 0,Y 467.512,Z 335.875,A -85,B 0,C 180,E1 -7523.036,E2 -7523.036} C_VEL
LIN {X 0,Y 467.554,Z 335.865,A -85,B 0,C 180,E1 -7526.209,E2 -7526.209} C_VEL
LIN {X 0,Y 467.55,Z 335.868,A -85,B 0,C 180,E1 -7529.265,E2 -7529.265} C_VEL
LIN {X 0,Y 467.536,Z 335.869,A -85,B 0,C 180,E1 -7532.48,E2 -7532.48} C_VEL
LIN {X 0,Y 467.542,Z 335.869,A -85,B 0,C 180,E1 -7535.109,E2 -7535.109} C_VEL
LIN {X 0,Y 467.519,Z 335.87,A -85,B 0,C 180,E1 -7537.925,E2 -7537.925} C_VEL
LIN {X 0,Y 467.605,Z 335.853,A -85,B 0,C 180,E1 -7540.691,E2 -7540.691} C_VEL
LIN {X 0,Y 467.622,Z 335.86,A -85,B 0,C 180,E1 -7544.304,E2 -7544.304} C_VEL
LIN {X 0,Y 467.64,Z 335.854,A -85,B 0,C 180,E1 -7547.854,E2 -7547.854} C_VEL
LIN {X 0,Y 467.649,Z 335.852,A -85,B 0,C 180,E1 -7551.357,E2 -7551.357} C_VEL
LIN {X 0,Y 467.677,Z 335.851,A -85,B 0,C 180,E1 -7553.962,E2 -7553.962} C_VEL
LIN {X 0,Y 467.806,Z 335.834,A -85,B 0,C 180,E1 -7557.417,E2 -7557.417} C_VEL
LIN {X 0,Y 467.831,Z 335.829,A -85,B 0,C 180,E1 -7560,E2 -7560} C_VEL
LIN {X 0,Y 467.802,Z 335.841,A -85,B 0,C 180,E1 -7562.583,E2 -7562.583} C_VEL
LIN {X 0,Y 467.693,Z 335.85,A -85,B 0,C 180,E1 -7566.038,E2 -7566.038} C_VEL
LIN {X 0,Y 467.617,Z 335.861,A -85,B 0,C 180,E1 -7568.644,E2 -7568.644} C_VEL
LIN {X 0,Y 467.631,Z 335.859,A -85,B 0,C 180,E1 -7572.146,E2 -7572.146} C_VEL
LIN {X 0,Y 467.623,Z 335.857,A -85,B 0,C 180,E1 -7575.696,E2 -7575.696} C_VEL
LIN {X 0,Y 467.605,Z 335.859,A -85,B 0,C 180,E1 -7579.309,E2 -7579.309} C_VEL
LIN {X 0,Y 467.516,Z 335.866,A -85,B 0,C 180,E1 -7582.075,E2 -7582.075} C_VEL
LIN {X 0,Y 467.54,Z 335.869,A -85,B 0,C 180,E1 -7584.891,E2 -7584.891} C_VEL
LIN {X 0,Y 467.532,Z 335.867,A -85,B 0,C 180,E1 -7587.775,E2 -7587.775} C_VEL
LIN {X 0,Y 467.533,Z 335.869,A -85,B 0,C 180,E1 -7591.041,E2 -7591.041} C_VEL
LIN {X 0,Y 467.562,Z 335.87,A -85,B 0,C 180,E1 -7594.241,E2 -7594.241} C_VEL
LIN {X 0,Y 467.502,Z 335.873,A -85,B 0,C 180,E1 -7597.182,E2 -7597.182} C_VEL
LIN {X 0,Y 467.526,Z 335.876,A -85,B 0,C 180,E1 -7600.27,E2 -7600.27} C_VEL
LIN {X 0,Y 467.504,Z 335.876,A -85,B 0,C 180,E1 -7602.57,E2 -7602.57} C_VEL
LIN {X 0,Y 467.55,Z 335.867,A -85,B 0,C 180,E1 -7605.053,E2 -7605.053} C_VEL
LIN {X 0,Y 467.539,Z 335.871,A -85,B 0,C 180,E1 -7608.729,E2 -7608.729} C_VEL
LIN {X 0,Y 467.527,Z 335.876,A -85,B 0,C 180,E1 -7611.954,E2 -7611.954} C_VEL
LIN {X 0,Y 467.541,Z 335.869,A -85,B 0,C 180,E1 -7615.167,E2 -7615.167} C_VEL
LIN {X 0,Y 467.547,Z 335.873,A -85,B 0,C 180,E1 -7618.259,E2 -7618.259} C_VEL
LIN {X 0,Y 467.535,Z 335.868,A -85,B 0,C 180,E1 -7621.25,E2 -7621.25} C_VEL
LIN {X 0,Y 467.574,Z 335.962,A -85,B 0,C 180,E1 -7623.118,E2 -7623.118} C_VEL
LIN {X 0,Y 470.458,Z 349.512,A -85,B 0,C 180,E1 -7625.68,E2 -7625.68} C_VEL
LIN {X 0,Y 470.528,Z 353.927,A -85,B 0,C 180,E1 -7626.452,E2 -7626.452} C_VEL
LIN {X 0,Y 469.659,Z 371.106,A -85,B 0,C 180,E1 -7629.367,E2 -7629.367} C_VEL
LIN {X 0,Y 473.398,Z 390.861,A -85,B 0,C 180,E1 -7629.863,E2 -7629.863} C_VEL
LIN {X 0,Y 472.431,Z 500.222,A -85,B 0,C 180,E1 -7631.545,E2 -7631.545} C_VEL
LIN {X 0,Y 472.117,Z 515.109,A -85,B 0,C 180,E1 -7631.847,E2 -7631.847} C_VEL
LIN {X 0,Y 471.674,Z 529.163,A -85,B 0,C 180,E1 -7632.311,E2 -7632.311} C_VEL
LIN {X 0,Y 471.107,Z 542.884,A -85,B 0,C 180,E1 -7632.946,E2 -7632.946} C_VEL
LIN {X 0,Y 470.477,Z 555.951,A -85,B 0,C 180,E1 -7633.736,E2 -7633.736} C_VEL
LIN {X 0,Y 469.729,Z 568.747,A -85,B 0,C 180,E1 -7634.712,E2 -7634.712} C_VEL
LIN {X 0,Y 469.038,Z 580.282,A -85,B 0,C 180,E1 -7635.798,E2 -7635.798} C_VEL
LIN {X 0,Y 468.425,Z 590.736,A -85,B 0,C 180,E1 -7636.996,E2 -7636.996} C_VEL
LIN {X 0,Y 467.956,Z 600.179,A -85,B 0,C 180,E1 -7638.304,E2 -7638.304} C_VEL
LIN {X 0,Y 467.38,Z 609.175,A -85,B 0,C 180,E1 -7639.825,E2 -7639.825} C_VEL
LIN {X 0,Y 467.074,Z 616.44,A -85,B 0,C 180,E1 -7641.347,E2 -7641.347} C_VEL
LIN {X 0,Y 466.831,Z 622.968,A -85,B 0,C 180,E1 -7643.084,E2 -7643.084} C_VEL
LIN {X 0,Y 466.764,Z 627.859,A -85,B 0,C 180,E1 -7644.818,E2 -7644.818} C_VEL
LIN {X 0,Y 466.651,Z 631.256,A -85,B 0,C 180,E1 -7646.548,E2 -7646.548} C_VEL
LIN {X 0,Y 466.601,Z 633.262,A -85,B 0,C 180,E1 -7648.275,E2 -7648.275} C_VEL
LIN {X 0,Y 466.597,Z 633.925,A -85,B 0,C 180,E1 -7650.001,E2 -7650.001} C_VEL
LIN {X 0,Y 466.601,Z 633.257,A -85,B 0,C 180,E1 -7651.728,E2 -7651.728} C_VEL
LIN {X 0,Y 466.651,Z 631.247,A -85,B 0,C 180,E1 -7653.455,E2 -7653.455} C_VEL
LIN {X 0,Y 466.763,Z 627.848,A -85,B 0,C 180,E1 -7655.184,E2 -7655.184} C_VEL
LIN {X 0,Y 466.825,Z 622.959,A -85,B 0,C 180,E1 -7656.919,E2 -7656.919} C_VEL
LIN {X 0,Y 467.077,Z 616.427,A -85,B 0,C 180,E1 -7658.655,E2 -7658.655} C_VEL
LIN {X 0,Y 467.385,Z 609.157,A -85,B 0,C 180,E1 -7660.178,E2 -7660.178} C_VEL
LIN {X 0,Y 467.973,Z 600.157,A -85,B 0,C 180,E1 -7661.699,E2 -7661.699} C_VEL
LIN {X 0,Y 468.434,Z 590.707,A -85,B 0,C 180,E1 -7663.007,E2 -7663.007} C_VEL
LIN {X 0,Y 469.055,Z 580.248,A -85,B 0,C 180,E1 -7664.204,E2 -7664.204} C_VEL
LIN {X 0,Y 469.764,Z 568.702,A -85,B 0,C 180,E1 -7665.29,E2 -7665.29} C_VEL
LIN {X 0,Y 470.489,Z 555.892,A -85,B 0,C 180,E1 -7666.266,E2 -7666.266} C_VEL
LIN {X 0,Y 471.155,Z 542.562,A -85,B 0,C 180,E1 -7667.069,E2 -7667.069} C_VEL
LIN {X 0,Y 471.649,Z 529.08,A -85,B 0,C 180,E1 -7667.692,E2 -7667.692} C_VEL
LIN {X 0,Y 472.156,Z 514.965,A -85,B 0,C 180,E1 -7668.154,E2 -7668.154} C_VEL
LIN {X 0,Y 472.388,Z 499.952,A -85,B 0,C 180,E1 -7668.459,E2 -7668.459} C_VEL
LIN {X 0,Y 473.437,Z 391.203,A -85,B 0,C 180,E1 -7670.128,E2 -7670.128} C_VEL
LIN {X 0,Y 469.637,Z 371.075,A -85,B 0,C 180,E1 -7670.637,E2 -7670.637} C_VEL
LIN {X 0,Y 470.598,Z 352.549,A -85,B 0,C 180,E1 -7673.781,E2 -7673.781} C_VEL
LIN {X 0,Y 470.299,Z 348.763,A -85,B 0,C 180,E1 -7674.456,E2 -7674.456} C_VEL
LIN {X 0,Y 467.57,Z 335.87,A -85,B 0,C 180,E1 -7676.913,E2 -7676.913} C_VEL
LIN {X 0,Y 467.545,Z 335.872,A -85,B 0,C 180,E1 -7679.74,E2 -7679.74} C_VEL
LIN {X 0,Y 467.588,Z 335.865,A -85,B 0,C 180,E1 -7682.759,E2 -7682.759} C_VEL
LIN {X 0,Y 467.556,Z 335.867,A -85,B 0,C 180,E1 -7685.891,E2 -7685.891} C_VEL
LIN {X 0,Y 467.58,Z 335.868,A -85,B 0,C 180,E1 -7689.146,E2 -7689.146} C_VEL
LIN {X 0,Y 467.592,Z 335.863,A -85,B 0,C 180,E1 -7692.568,E2 -7692.568} C_VEL
LIN {X 0,Y 467.576,Z 335.87,A -85,B 0,C 180,E1 -7695.054,E2 -7695.054} C_VEL
LIN {X 0,Y 467.594,Z 335.863,A -85,B 0,C 180,E1 -7697.44,E2 -7697.44} C_VEL
LIN {X 0,Y 467.586,Z 335.867,A -85,B 0,C 180,E1 -7700.856,E2 -7700.856} C_VEL
LIN {X 0,Y 467.562,Z 335.87,A -85,B 0,C 180,E1 -7704.262,E2 -7704.262} C_VEL
LIN {X 0,Y 467.587,Z 335.865,A -85,B 0,C 180,E1 -7707.321,E2 -7707.321} C_VEL
LIN {X 0,Y 467.562,Z 335.874,A -85,B 0,C 180,E1 -7710.671,E2 -7710.671} C_VEL
LIN {X 0,Y 467.556,Z 335.873,A -85,B 0,C 180,E1 -7713.196,E2 -7713.196} C_VEL
LIN {X 0,Y 467.611,Z 335.994,A -85,B 0,C 180,E1 -7715.97,E2 -7715.97} C_VEL
LIN {X 0,Y 469.662,Z 346.295,A -85,B 0,C 180,E1 -7717.8,E2 -7717.8} C_VEL
LIN {X 0,Y 469.509,Z 361.608,A -85,B 0,C 180,E1 -7720.364,E2 -7720.364} C_VEL
LIN {X 0,Y 469.145,Z 377.42,A -85,B 0,C 180,E1 -7722.994,E2 -7722.994} C_VEL
LIN {X 0,Y 471.472,Z 389.527,A -85,B 0,C 180,E1 -7723.334,E2 -7723.334} C_VEL
LIN {X 0,Y 470.192,Z 487.239,A -85,B 0,C 180,E1 -7725.114,E2 -7725.114} C_VEL
LIN {X 0,Y 469.894,Z 500.612,A -85,B 0,C 180,E1 -7725.547,E2 -7725.547} C_VEL
LIN {X 0,Y 469.539,Z 513.432,A -85,B 0,C 180,E1 -7726.144,E2 -7726.144} C_VEL
LIN {X 0,Y 469.105,Z 525.688,A -85,B 0,C 180,E1 -7726.914,E2 -7726.914} C_VEL
LIN {X 0,Y 468.791,Z 536.439,A -85,B 0,C 180,E1 -7727.777,E2 -7727.777} C_VEL
LIN {X 0,Y 468.283,Z 546.307,A -85,B 0,C 180,E1 -7728.749,E2 -7728.749} C_VEL
LIN {X 0,Y 467.901,Z 555.216,A -85,B 0,C 180,E1 -7729.835,E2 -7729.835} C_VEL
LIN {X 0,Y 467.501,Z 563.907,A -85,B 0,C 180,E1 -7731.136,E2 -7731.136} C_VEL
LIN {X 0,Y 467.225,Z 570.849,A -85,B 0,C 180,E1 -7732.437,E2 -7732.437} C_VEL
LIN {X 0,Y 467.05,Z 577.144,A -85,B 0,C 180,E1 -7733.954,E2 -7733.954} C_VEL
LIN {X 0,Y 466.847,Z 581.249,A -85,B 0,C 180,E1 -7735.251,E2 -7735.251} C_VEL
LIN {X 0,Y 466.819,Z 584.264,A -85,B 0,C 180,E1 -7736.548,E2 -7736.548} C_VEL
LIN {X 0,Y 466.75,Z 585.739,A -85,B 0,C 180,E1 -7737.411,E2 -7737.411} C_VEL
LIN {X 0,Y 466.698,Z 586.75,A -85,B 0,C 180,E1 -7738.274,E2 -7738.274} C_VEL
LIN {X 0,Y 466.604,Z 587.583,A -85,B 0,C 180,E1 -7740,E2 -7740} C_VEL
LIN {X 0,Y 466.623,Z 587.352,A -85,B 0,C 180,E1 -7740.863,E2 -7740.863} C_VEL
LIN {X 0,Y 466.697,Z 586.709,A -85,B 0,C 180,E1 -7741.726,E2 -7741.726} C_VEL
LIN {X 0,Y 466.732,Z 585.674,A -85,B 0,C 180,E1 -7742.589,E2 -7742.589} C_VEL
LIN {X 0,Y 466.797,Z 584.204,A -85,B 0,C 180,E1 -7743.453,E2 -7743.453} C_VEL
LIN {X 0,Y 466.789,Z 581.169,A -85,B 0,C 180,E1 -7744.75,E2 -7744.75} C_VEL
LIN {X 0,Y 467.04,Z 577.048,A -85,B 0,C 180,E1 -7746.047,E2 -7746.047} C_VEL
LIN {X 0,Y 467.14,Z 570.734,A -85,B 0,C 180,E1 -7747.565,E2 -7747.565} C_VEL
LIN {X 0,Y 467.456,Z 563.83,A -85,B 0,C 180,E1 -7748.865,E2 -7748.865} C_VEL
LIN {X 0,Y 467.806,Z 555.152,A -85,B 0,C 180,E1 -7750.167,E2 -7750.167} C_VEL
LIN {X 0,Y 468.245,Z 545.298,A -85,B 0,C 180,E1 -7751.361,E2 -7751.361} C_VEL
LIN {X 0,Y 468.746,Z 534.352,A -85,B 0,C 180,E1 -7752.417,E2 -7752.417} C_VEL
LIN {X 0,Y 469.07,Z 523.303,A -85,B 0,C 180,E1 -7753.275,E2 -7753.275} C_VEL
LIN {X 0,Y 469.506,Z 510.807,A -85,B 0,C 180,E1 -7754.023,E2 -7754.023} C_VEL
LIN {X 0,Y 469.855,Z 498.745,A -85,B 0,C 180,E1 -7754.565,E2 -7754.565} C_VEL
LIN {X 0,Y 470.164,Z 485.711,A -85,B 0,C 180,E1 -7754.97,E2 -7754.97} C_VEL
LIN {X 0,Y 470.505,Z 454.936,A -85,B 0,C 180,E1 -7755.514,E2 -7755.514} C_VEL
LIN {X 0,Y 471.077,Z 388.949,A -85,B 0,C 180,E1 -7756.643,E2 -7756.643} C_VEL
LIN {X 0,Y 468.692,Z 375.5,A -85,B 0,C 180,E1 -7756.985,E2 -7756.985} C_VEL
LIN {X 0,Y 469.165,Z 358.577,A -85,B 0,C 180,E1 -7759.925,E2 -7759.925} C_VEL
LIN {X 0,Y 469.376,Z 345.42,A -85,B 0,C 180,E1 -7762.214,E2 -7762.214} C_VEL
LIN {X 0,Y 467.608,Z 335.866,A -85,B 0,C 180,E1 -7764,E2 -7764} C_VEL
LIN {X 0,Y 467.618,Z 335.861,A -85,B 0,C 180,E1 -7766.8,E2 -7766.8} C_VEL
LIN {X 0,Y 467.559,Z 335.868,A -85,B 0,C 180,E1 -7769.738,E2 -7769.738} C_VEL
LIN {X 0,Y 467.589,Z 335.862,A -85,B 0,C 180,E1 -7772.758,E2 -7772.758} C_VEL
LIN {X 0,Y 467.556,Z 335.872,A -85,B 0,C 180,E1 -7775.89,E2 -7775.89} C_VEL
LIN {X 0,Y 467.557,Z 335.866,A -85,B 0,C 180,E1 -7779.147,E2 -7779.147} C_VEL
LIN {X 0,Y 467.572,Z 335.866,A -85,B 0,C 180,E1 -7781.404,E2 -7781.404} C_VEL
LIN {X 0,Y 467.571,Z 335.865,A -85,B 0,C 180,E1 -7784.947,E2 -7784.947} C_VEL
LIN {X 0,Y 467.569,Z 335.864,A -85,B 0,C 180,E1 -7788.595,E2 -7788.595} C_VEL
LIN {X 0,Y 467.547,Z 335.874,A -85,B 0,C 180,E1 -7791.412,E2 -7791.412} C_VEL
LIN {X 0,Y 467.56,Z 335.866,A -85,B 0,C 180,E1 -7794.261,E2 -7794.261} C_VEL
LIN {X 0,Y 467.551,Z 335.871,A -85,B 0,C 180,E1 -7797.327,E2 -7797.327} C_VEL
LIN {X 0,Y 467.53,Z 335.871,A -85,B 0,C 180,E1 -7800.088,E2 -7800.088} C_VEL
LIN {X 0,Y 466.884,Z 335.955,A -85,B 0,C 180,E1 -7800.808,E2 -7800.808} C_VEL
LIN {X 0,Y 464.04,Z 336.307,A -85,B 0,C 180,E1 -7801.976,E2 -7801.976} C_VEL
LIN {X 0,Y 461.624,Z 336.605,A -85,B 0,C 180,E1 -7802.918,E2 -7802.918} C_VEL
LIN {X 0,Y 460.589,Z 336.736,A -85,B 0,C 180,E1 -7803.646,E2 -7803.646} C_VEL
LIN {X 0,Y 460.507,Z 336.749,A -85,B 0,C 180,E1 -7803.893,E2 -7803.893} C_VEL
LIN {X 0,Y 460.568,Z 336.981,A -85,B 0,C 180,E1 -7804.091,E2 -7804.091} C_VEL
LIN {X 0,Y 463.333,Z 350.342,A -85,B 0,C 180,E1 -7806.772,E2 -7806.772} C_VEL
LIN {X 0,Y 463.098,Z 358.103,A -85,B 0,C 180,E1 -7808.193,E2 -7808.193} C_VEL
LIN {X 0,Y 462.85,Z 363.396,A -85,B 0,C 180,E1 -7809.119,E2 -7809.119} C_VEL
LIN {X 0,Y 466.875,Z 383.665,A -85,B 0,C 180,E1 -7809.635,E2 -7809.635} C_VEL
LIN {X 0,Y 465.584,Z 499.927,A -85,B 0,C 180,E1 -7811.461,E2 -7811.461} C_VEL
LIN {X 0,Y 465.184,Z 514.009,A -85,B 0,C 180,E1 -7811.846,E2 -7811.846} C_VEL
LIN {X 0,Y 464.734,Z 527.575,A -85,B 0,C 180,E1 -7812.394,E2 -7812.394} C_VEL
LIN {X 0,Y 464.142,Z 540.21,A -85,B 0,C 180,E1 -7813.07,E2 -7813.07} C_VEL
LIN {X 0,Y 463.449,Z 552.862,A -85,B 0,C 180,E1 -7813.932,E2 -7813.932} C_VEL
LIN {X 0,Y 462.711,Z 564.587,A -85,B 0,C 180,E1 -7814.922,E2 -7814.922} C_VEL
LIN {X 0,Y 461.932,Z 576.283,A -85,B 0,C 180,E1 -7816.134,E2 -7816.134} C_VEL
LIN {X 0,Y 461.413,Z 585.488,A -85,B 0,C 180,E1 -7817.292,E2 -7817.292} C_VEL
LIN {X 0,Y 460.891,Z 593.996,A -85,B 0,C 180,E1 -7818.565,E2 -7818.565} C_VEL
LIN {X 0,Y 460.409,Z 602.505,A -85,B 0,C 180,E1 -7820.11,E2 -7820.11} C_VEL
LIN {X 0,Y 460.044,Z 609.364,A -85,B 0,C 180,E1 -7821.654,E2 -7821.654} C_VEL
LIN {X 0,Y 459.84,Z 614.099,A -85,B 0,C 180,E1 -7822.976,E2 -7822.976} C_VEL
LIN {X 0,Y 459.709,Z 618.998,A -85,B 0,C 180,E1 -7824.736,E2 -7824.736} C_VEL
LIN {X 0,Y 459.59,Z 622.413,A -85,B 0,C 180,E1 -7826.492,E2 -7826.492} C_VEL
LIN {X 0,Y 459.519,Z 624.446,A -85,B 0,C 180,E1 -7828.246,E2 -7828.246} C_VEL
LIN {X 0,Y 459.5,Z 625.148,A -85,B 0,C 180,E1 -7829.999,E2 -7829.999} C_VEL
LIN {X 0,Y 459.518,Z 624.528,A -85,B 0,C 180,E1 -7831.752,E2 -7831.752} C_VEL
LIN {X 0,Y 459.589,Z 622.571,A -85,B 0,C 180,E1 -7833.505,E2 -7833.505} C_VEL
LIN {X 0,Y 459.708,Z 619.227,A -85,B 0,C 180,E1 -7835.262,E2 -7835.262} C_VEL
LIN {X 0,Y 459.837,Z 614.399,A -85,B 0,C 180,E1 -7837.022,E2 -7837.022} C_VEL
LIN {X 0,Y 460.094,Z 607.941,A -85,B 0,C 180,E1 -7838.785,E2 -7838.785} C_VEL
LIN {X 0,Y 460.458,Z 600.751,A -85,B 0,C 180,E1 -7840.33,E2 -7840.33} C_VEL
LIN {X 0,Y 461.036,Z 591.856,A -85,B 0,C 180,E1 -7841.874,E2 -7841.874} C_VEL
LIN {X 0,Y 461.586,Z 582.513,A -85,B 0,C 180,E1 -7843.201,E2 -7843.201} C_VEL
LIN {X 0,Y 462.225,Z 572.162,A -85,B 0,C 180,E1 -7844.415,E2 -7844.415} C_VEL
LIN {X 0,Y 462.957,Z 560.745,A -85,B 0,C 180,E1 -7845.518,E2 -7845.518} C_VEL
LIN {X 0,Y 463.742,Z 548.091,A -85,B 0,C 180,E1 -7846.507,E2 -7846.507} C_VEL
LIN {X 0,Y 464.373,Z 535.18,A -85,B 0,C 180,E1 -7847.311,E2 -7847.311} C_VEL
LIN {X 0,Y 464.951,Z 522.148,A -85,B 0,C 180,E1 -7847.935,E2 -7847.935} C_VEL
LIN {X 0,Y 465.424,Z 507.967,A -85,B 0,C 180,E1 -7848.429,E2 -7848.429} C_VEL
LIN {X 0,Y 465.705,Z 494.447,A -85,B 0,C 180,E1 -7848.731,E2 -7848.731} C_VEL
LIN {X 0,Y 466.885,Z 383.54,A -85,B 0,C 180,E1 -7850.459,E2 -7850.459} C_VEL
LIN {X 0,Y 462.828,Z 363.16,A -85,B 0,C 180,E1 -7850.988,E2 -7850.988} C_VEL
LIN {X 0,Y 463.365,Z 350.862,A -85,B 0,C 180,E1 -7853.224,E2 -7853.224} C_VEL
LIN {X 0,Y 461.13,Z 339.629,A -85,B 0,C 180,E1 -7855.464,E2 -7855.464} C_VEL
LIN {X 0,Y 460.507,Z 336.749,A -85,B 0,C 180,E1 -7856.056,E2 -7856.056} C_VEL
LIN {X 0,Y 460.51,Z 336.752,A -85,B 0,C 180,E1 -7859.231,E2 -7859.231} C_VEL
LIN {X 0,Y 460.515,Z 336.748,A -85,B 0,C 180,E1 -7862.284,E2 -7862.284} C_VEL
LIN {X 0,Y 460.499,Z 336.749,A -85,B 0,C 180,E1 -7865.445,E2 -7865.445} C_VEL
LIN {X 0,Y 460.491,Z 336.752,A -85,B 0,C 180,E1 -7868.889,E2 -7868.889} C_VEL
LIN {X 0,Y 460.493,Z 336.746,A -85,B 0,C 180,E1 -7871.597,E2 -7871.597} C_VEL
LIN {X 0,Y 460.501,Z 336.748,A -85,B 0,C 180,E1 -7874.588,E2 -7874.588} C_VEL
LIN {X 0,Y 460.469,Z 336.748,A -85,B 0,C 180,E1 -7877.812,E2 -7877.812} C_VEL
LIN {X 0,Y 460.502,Z 336.745,A -85,B 0,C 180,E1 -7880.134,E2 -7880.134} C_VEL
LIN {X 0,Y 460.46,Z 336.75,A -85,B 0,C 180,E1 -7883.469,E2 -7883.469} C_VEL
LIN {X 0,Y 460.504,Z 336.743,A -85,B 0,C 180,E1 -7886.673,E2 -7886.673} C_VEL
LIN {X 0,Y 460.489,Z 336.745,A -85,B 0,C 180,E1 -7889.758,E2 -7889.758} C_VEL
LIN {X 0,Y 460.476,Z 336.743,A -85,B 0,C 180,E1 -7892.75,E2 -7892.75} C_VEL
LIN {X 0,Y 460.502,Z 336.742,A -85,B 0,C 180,E1 -7895.665,E2 -7895.665} C_VEL
LIN {X 0,Y 460.507,Z 336.747,A -85,B 0,C 180,E1 -7898.578,E2 -7898.578} C_VEL
LIN {X 0,Y 460.569,Z 336.728,A -85,B 0,C 180,E1 -7901.31,E2 -7901.31} C_VEL
LIN {X 0,Y 460.571,Z 336.736,A -85,B 0,C 180,E1 -7904.058,E2 -7904.058} C_VEL
LIN {X 0,Y 460.594,Z 336.731,A -85,B 0,C 180,E1 -7907.665,E2 -7907.665} C_VEL
LIN {X 0,Y 460.6,Z 336.731,A -85,B 0,C 180,E1 -7911.223,E2 -7911.223} C_VEL
LIN {X 0,Y 460.644,Z 336.727,A -85,B 0,C 180,E1 -7913.869,E2 -7913.869} C_VEL
LIN {X 0,Y 460.75,Z 336.713,A -85,B 0,C 180,E1 -7917.377,E2 -7917.377} C_VEL
LIN {X 0,Y 460.78,Z 336.708,A -85,B 0,C 180,E1 -7920,E2 -7920} C_VEL
LIN {X 0,Y 460.746,Z 336.719,A -85,B 0,C 180,E1 -7922.623,E2 -7922.623} C_VEL
LIN {X 0,Y 460.658,Z 336.727,A -85,B 0,C 180,E1 -7926.131,E2 -7926.131} C_VEL
LIN {X 0,Y 460.572,Z 336.738,A -85,B 0,C 180,E1 -7928.777,E2 -7928.777} C_VEL
LIN {X 0,Y 460.581,Z 336.738,A -85,B 0,C 180,E1 -7932.435,E2 -7932.435} C_VEL
LIN {X 0,Y 460.586,Z 336.736,A -85,B 0,C 180,E1 -7935.998,E2 -7935.998} C_VEL
LIN {X 0,Y 460.552,Z 336.737,A -85,B 0,C 180,E1 -7939.616,E2 -7939.616} C_VEL
LIN {X 0,Y 460.493,Z 336.74,A -85,B 0,C 180,E1 -7942.43,E2 -7942.43} C_VEL
LIN {X 0,Y 460.518,Z 336.743,A -85,B 0,C 180,E1 -7945.793,E2 -7945.793} C_VEL
LIN {X 0,Y 460.507,Z 336.736,A -85,B 0,C 180,E1 -7949.233,E2 -7949.233} C_VEL
LIN {X 0,Y 460.504,Z 336.751,A -85,B 0,C 180,E1 -7952.287,E2 -7952.287} C_VEL
LIN {X 0,Y 460.486,Z 336.746,A -85,B 0,C 180,E1 -7955.448,E2 -7955.448} C_VEL
LIN {X 0,Y 460.471,Z 336.75,A -85,B 0,C 180,E1 -7958.889,E2 -7958.889} C_VEL
LIN {X 0,Y 460.483,Z 336.747,A -85,B 0,C 180,E1 -7961.598,E2 -7961.598} C_VEL
LIN {X 0,Y 460.498,Z 336.749,A -85,B 0,C 180,E1 -7964.591,E2 -7964.591} C_VEL
LIN {X 0,Y 460.46,Z 336.754,A -85,B 0,C 180,E1 -7967.814,E2 -7967.814} C_VEL
LIN {X 0,Y 460.471,Z 336.75,A -85,B 0,C 180,E1 -7971.114,E2 -7971.114} C_VEL
LIN {X 0,Y 460.491,Z 336.751,A -85,B 0,C 180,E1 -7974.555,E2 -7974.555} C_VEL
LIN {X 0,Y 460.508,Z 336.748,A -85,B 0,C 180,E1 -7977.716,E2 -7977.716} C_VEL
LIN {X 0,Y 460.512,Z 336.742,A -85,B 0,C 180,E1 -7980.769,E2 -7980.769} C_VEL
LIN {X 0,Y 460.556,Z 336.859,A -85,B 0,C 180,E1 -7982.849,E2 -7982.849} C_VEL
LIN {X 0,Y 463.472,Z 350.537,A -85,B 0,C 180,E1 -7985.482,E2 -7985.482} C_VEL
LIN {X 0,Y 463.743,Z 353.867,A -85,B 0,C 180,E1 -7986.086,E2 -7986.086} C_VEL
LIN {X 0,Y 462.758,Z 371.091,A -85,B 0,C 180,E1 -7989.054,E2 -7989.054} C_VEL
LIN {X 0,Y 466.808,Z 392.844,A -85,B 0,C 180,E1 -7989.599,E2 -7989.599} C_VEL
LIN {X 0,Y 465.573,Z 507.945,A -85,B 0,C 180,E1 -7991.406,E2 -7991.406} C_VEL
LIN {X 0,Y 465.147,Z 522.103,A -85,B 0,C 180,E1 -7991.787,E2 -7991.787} C_VEL
LIN {X 0,Y 464.594,Z 535.811,A -85,B 0,C 180,E1 -7992.334,E2 -7992.334} C_VEL
LIN {X 0,Y 464.044,Z 548.345,A -85,B 0,C 180,E1 -7993.002,E2 -7993.002} C_VEL
LIN {X 0,Y 463.415,Z 560.5,A -85,B 0,C 180,E1 -7993.821,E2 -7993.821} C_VEL
LIN {X 0,Y 462.616,Z 572.39,A -85,B 0,C 180,E1 -7994.809,E2 -7994.809} C_VEL
LIN {X 0,Y 461.918,Z 583.253,A -85,B 0,C 180,E1 -7995.912,E2 -7995.912} C_VEL
LIN {X 0,Y 461.281,Z 593.604,A -85,B 0,C 180,E1 -7997.186,E2 -7997.186} C_VEL
LIN {X 0,Y 460.773,Z 602.851,A -85,B 0,C 180,E1 -7998.565,E2 -7998.565} C_VEL
LIN {X 0,Y 460.258,Z 611.344,A -85,B 0,C 180,E1 -8000.11,E2 -8000.11} C_VEL
LIN {X 0,Y 459.93,Z 618.185,A -85,B 0,C 180,E1 -8001.655,E2 -8001.655} C_VEL
LIN {X 0,Y 459.738,Z 622.901,A -85,B 0,C 180,E1 -8002.977,E2 -8002.977} C_VEL
LIN {X 0,Y 459.675,Z 627.792,A -85,B 0,C 180,E1 -8004.738,E2 -8004.738} C_VEL
LIN {X 0,Y 459.547,Z 631.189,A -85,B 0,C 180,E1 -8006.494,E2 -8006.494} C_VEL
LIN {X 0,Y 459.513,Z 633.195,A -85,B 0,C 180,E1 -8008.248,E2 -8008.248} C_VEL
LIN {X 0,Y 459.499,Z 633.858,A -85,B 0,C 180,E1 -8010.001,E2 -8010.001} C_VEL
LIN {X 0,Y 459.514,Z 633.19,A -85,B 0,C 180,E1 -8011.754,E2 -8011.754} C_VEL
LIN {X 0,Y 459.548,Z 631.179,A -85,B 0,C 180,E1 -8013.508,E2 -8013.508} C_VEL
LIN {X 0,Y 459.674,Z 627.78,A -85,B 0,C 180,E1 -8015.265,E2 -8015.265} C_VEL
LIN {X 0,Y 459.736,Z 622.891,A -85,B 0,C 180,E1 -8017.026,E2 -8017.026} C_VEL
LIN {X 0,Y 460.022,Z 616.358,A -85,B 0,C 180,E1 -8018.789,E2 -8018.789} C_VEL
LIN {X 0,Y 460.358,Z 609.088,A -85,B 0,C 180,E1 -8020.335,E2 -8020.335} C_VEL
LIN {X 0,Y 460.98,Z 600.088,A -85,B 0,C 180,E1 -8021.879,E2 -8021.879} C_VEL
LIN {X 0,Y 461.48,Z 590.637,A -85,B 0,C 180,E1 -8023.206,E2 -8023.206} C_VEL
LIN {X 0,Y 462.148,Z 580.178,A -85,B 0,C 180,E1 -8024.421,E2 -8024.421} C_VEL
LIN {X 0,Y 462.889,Z 568.632,A -85,B 0,C 180,E1 -8025.523,E2 -8025.523} C_VEL
LIN {X 0,Y 463.66,Z 555.821,A -85,B 0,C 180,E1 -8026.513,E2 -8026.513} C_VEL
LIN {X 0,Y 464.345,Z 543.094,A -85,B 0,C 180,E1 -8027.293,E2 -8027.293} C_VEL
LIN {X 0,Y 464.822,Z 530.179,A -85,B 0,C 180,E1 -8027.91,E2 -8027.91} C_VEL
LIN {X 0,Y 465.346,Z 516.939,A -85,B 0,C 180,E1 -8028.367,E2 -8028.367} C_VEL
LIN {X 0,Y 465.615,Z 503.187,A -85,B 0,C 180,E1 -8028.681,E2 -8028.681} C_VEL
LIN {X 0,Y 466.826,Z 392.588,A -85,B 0,C 180,E1 -8030.402,E2 -8030.402} C_VEL
LIN {X 0,Y 462.731,Z 371.01,A -85,B 0,C 180,E1 -8030.958,E2 -8030.958} C_VEL
LIN {X 0,Y 463.724,Z 353.83,A -85,B 0,C 180,E1 -8033.918,E2 -8033.918} C_VEL
LIN {X 0,Y 463.001,Z 348.175,A -85,B 0,C 180,E1 -8034.961,E2 -8034.961} C_VEL
LIN {X 0,Y 460.553,Z 336.745,A -85,B 0,C 180,E1 -8037.185,E2 -8037.185} C_VEL
LIN {X 0,Y 460.507,Z 336.747,A -85,B 0,C 180,E1 -8040.241,E2 -8040.241} C_VEL
LIN {X 0,Y 460.534,Z 336.745,A -85,B 0,C 180,E1 -8043.326,E2 -8043.326} C_VEL
LIN {X 0,Y 460.477,Z 336.749,A -85,B 0,C 180,E1 -8046.53,E2 -8046.53} C_VEL
LIN {X 0,Y 460.532,Z 336.741,A -85,B 0,C 180,E1 -8049.863,E2 -8049.863} C_VEL
LIN {X 0,Y 460.518,Z 336.747,A -85,B 0,C 180,E1 -8052.901,E2 -8052.901} C_VEL
LIN {X 0,Y 460.517,Z 336.744,A -85,B 0,C 180,E1 -8055.831,E2 -8055.831} C_VEL
LIN {X 0,Y 460.536,Z 336.745,A -85,B 0,C 180,E1 -8058.989,E2 -8058.989} C_VEL
LIN {X 0,Y 460.53,Z 336.742,A -85,B 0,C 180,E1 -8061.267,E2 -8061.267} C_VEL
LIN {X 0,Y 460.513,Z 336.748,A -85,B 0,C 180,E1 -8064.555,E2 -8064.555} C_VEL
LIN {X 0,Y 460.537,Z 336.745,A -85,B 0,C 180,E1 -8067.716,E2 -8067.716} C_VEL
LIN {X 0,Y 460.531,Z 336.749,A -85,B 0,C 180,E1 -8070.768,E2 -8070.768} C_VEL
LIN {X 0,Y 460.523,Z 336.75,A -85,B 0,C 180,E1 -8073.732,E2 -8073.732} C_VEL
LIN {X 0,Y 460.587,Z 336.93,A -85,B 0,C 180,E1 -8075.67,E2 -8075.67} C_VEL
LIN {X 0,Y 462.638,Z 346.677,A -85,B 0,C 180,E1 -8077.445,E2 -8077.445} C_VEL
LIN {X 0,Y 462.866,Z 351.393,A -85,B 0,C 180,E1 -8078.263,E2 -8078.263} C_VEL
LIN {X 0,Y 462.512,Z 368.671,A -85,B 0,C 180,E1 -8081.163,E2 -8081.163} C_VEL
LIN {X 0,Y 462.284,Z 377.589,A -85,B 0,C 180,E1 -8082.681,E2 -8082.681} C_VEL
LIN {X 0,Y 464.785,Z 390.274,A -85,B 0,C 180,E1 -8083.055,E2 -8083.055} C_VEL
LIN {X 0,Y 463.383,Z 486.651,A -85,B 0,C 180,E1 -8084.862,E2 -8084.862} C_VEL
LIN {X 0,Y 463.088,Z 499.727,A -85,B 0,C 180,E1 -8085.274,E2 -8085.274} C_VEL
LIN {X 0,Y 462.696,Z 512.796,A -85,B 0,C 180,E1 -8085.879,E2 -8085.879} C_VEL
LIN {X 0,Y 462.274,Z 524.712,A -85,B 0,C 180,E1 -8086.617,E2 -8086.617} C_VEL
LIN {X 0,Y 461.857,Z 536.873,A -85,B 0,C 180,E1 -8087.597,E2 -8087.597} C_VEL
LIN {X 0,Y 461.328,Z 546.66,A -85,B 0,C 180,E1 -8088.577,E2 -8088.577} C_VEL
LIN {X 0,Y 460.921,Z 555.58,A -85,B 0,C 180,E1 -8089.679,E2 -8089.679} C_VEL
LIN {X 0,Y 460.5,Z 564.27,A -85,B 0,C 180,E1 -8091,E2 -8091} C_VEL
LIN {X 0,Y 460.209,Z 571.209,A -85,B 0,C 180,E1 -8092.321,E2 -8092.321} C_VEL
LIN {X 0,Y 460.006,Z 577.504,A -85,B 0,C 180,E1 -8093.861,E2 -8093.861} C_VEL
LIN {X 0,Y 459.762,Z 581.61,A -85,B 0,C 180,E1 -8095.177,E2 -8095.177} C_VEL
LIN {X 0,Y 459.754,Z 584.623,A -85,B 0,C 180,E1 -8096.494,E2 -8096.494} C_VEL
LIN {X 0,Y 459.67,Z 586.091,A -85,B 0,C 180,E1 -8097.371,E2 -8097.371} C_VEL
LIN {X 0,Y 459.636,Z 587.094,A -85,B 0,C 180,E1 -8098.248,E2 -8098.248} C_VEL
LIN {X 0,Y 459.556,Z 587.703,A -85,B 0,C 180,E1 -8099.124,E2 -8099.124} C_VEL
LIN {X 0,Y 459.535,Z 587.912,A -85,B 0,C 180,E1 -8100,E2 -8100} C_VEL
LIN {X 0,Y 459.556,Z 587.665,A -85,B 0,C 180,E1 -8100.876,E2 -8100.876} C_VEL
LIN {X 0,Y 459.605,Z 587.013,A -85,B 0,C 180,E1 -8101.753,E2 -8101.753} C_VEL
LIN {X 0,Y 459.652,Z 585.964,A -85,B 0,C 180,E1 -8102.629,E2 -8102.629} C_VEL
LIN {X 0,Y 459.732,Z 584.47,A -85,B 0,C 180,E1 -8103.506,E2 -8103.506} C_VEL
LIN {X 0,Y 459.708,Z 581.403,A -85,B 0,C 180,E1 -8104.823,E2 -8104.823} C_VEL
LIN {X 0,Y 459.974,Z 576.209,A -85,B 0,C 180,E1 -8106.422,E2 -8106.422} C_VEL
LIN {X 0,Y 460.136,Z 569.828,A -85,B 0,C 180,E1 -8107.901,E2 -8107.901} C_VEL
LIN {X 0,Y 460.481,Z 562.567,A -85,B 0,C 180,E1 -8109.222,E2 -8109.222} C_VEL
LIN {X 0,Y 460.863,Z 553.538,A -85,B 0,C 180,E1 -8110.544,E2 -8110.544} C_VEL
LIN {X 0,Y 461.361,Z 543.117,A -85,B 0,C 180,E1 -8111.756,E2 -8111.756} C_VEL
LIN {X 0,Y 461.814,Z 533.453,A -85,B 0,C 180,E1 -8112.67,E2 -8112.67} C_VEL
LIN {X 0,Y 462.165,Z 522.326,A -85,B 0,C 180,E1 -8113.521,E2 -8113.521} C_VEL
LIN {X 0,Y 462.644,Z 509.22,A -85,B 0,C 180,E1 -8114.291,E2 -8114.291} C_VEL
LIN {X 0,Y 462.971,Z 496.411,A -85,B 0,C 180,E1 -8114.843,E2 -8114.843} C_VEL
LIN {X 0,Y 463.296,Z 483.002,A -85,B 0,C 180,E1 -8115.226,E2 -8115.226} C_VEL
LIN {X 0,Y 464.271,Z 390.055,A -85,B 0,C 180,E1 -8116.855,E2 -8116.855} C_VEL
LIN {X 0,Y 461.751,Z 375.831,A -85,B 0,C 180,E1 -8117.209,E2 -8117.209} C_VEL
LIN {X 0,Y 462.219,Z 358.481,A -85,B 0,C 180,E1 -8120.238,E2 -8120.238} C_VEL
LIN {X 0,Y 462.508,Z 348.191,A -85,B 0,C 180,E1 -8122.038,E2 -8122.038} C_VEL
LIN {X 0,Y 461.101,Z 339.353,A -85,B 0,C 180,E1 -8123.667,E2 -8123.667} C_VEL
LIN {X 0,Y 460.568,Z 336.743,A -85,B 0,C 180,E1 -8124.172,E2 -8124.172} C_VEL
LIN {X 0,Y 460.576,Z 336.737,A -85,B 0,C 180,E1 -8127.244,E2 -8127.244} C_VEL
LIN {X 0,Y 460.516,Z 336.747,A -85,B 0,C 180,E1 -8130.24,E2 -8130.24} C_VEL
LIN {X 0,Y 460.535,Z 336.741,A -85,B 0,C 180,E1 -8133.325,E2 -8133.325} C_VEL
LIN {X 0,Y 460.478,Z 336.749,A -85,B 0,C 180,E1 -8136.529,E2 -8136.529} C_VEL
LIN {X 0,Y 460.519,Z 336.75,A -85,B 0,C 180,E1 -8139.864,E2 -8139.864} C_VEL
LIN {X 0,Y 460.497,Z 336.745,A -85,B 0,C 180,E1 -8142.897,E2 -8142.897} C_VEL
LIN {X 0,Y 460.509,Z 336.75,A -85,B 0,C 180,E1 -8145.831,E2 -8145.831} C_VEL
LIN {X 0,Y 460.523,Z 336.743,A -85,B 0,C 180,E1 -8148.987,E2 -8148.987} C_VEL
LIN {X 0,Y 460.491,Z 336.747,A -85,B 0,C 180,E1 -8152.375,E2 -8152.375} C_VEL
LIN {X 0,Y 460.539,Z 336.744,A -85,B 0,C 180,E1 -8155.622,E2 -8155.622} C_VEL
LIN {X 0,Y 460.509,Z 336.748,A -85,B 0,C 180,E1 -8158.741,E2 -8158.741} C_VEL
LIN {X 0,Y 460.507,Z 336.748,A -85,B 0,C 180,E1 -8161.763,E2 -8161.763} C_VEL
LIN {X 0,Y 460.507,Z 336.749,A -85,B 0,C 180,E1 -8163.893,E2 -8163.893} C_VEL
LIN {X 0,Y 460.466,Z 337.353,A -85,B 0,C 180,E1 -8164.149,E2 -8164.149} C_VEL
LIN {X 0,Y 459.955,Z 340.961,A -85,B 0,C 180,E1 -8164.813,E2 -8164.813} C_VEL
LIN {X 0,Y 457.383,Z 350.094,A -85,B 0,C 180,E1 -8166.352,E2 -8166.352} C_VEL
LIN {X 0,Y 456.526,Z 354.344,A -85,B 0,C 180,E1 -8167.147,E2 -8167.147} C_VEL
LIN {X 0,Y 456.015,Z 363.453,A -85,B 0,C 180,E1 -8168.79,E2 -8168.79} C_VEL
LIN {X 0,Y 460.133,Z 383.732,A -85,B 0,C 180,E1 -8169.322,E2 -8169.322} C_VEL
LIN {X 0,Y 459.242,Z 472.694,A -85,B 0,C 180,E1 -8170.731,E2 -8170.731} C_VEL
LIN {X 0,Y 458.855,Z 501.184,A -85,B 0,C 180,E1 -8171.208,E2 -8171.208} C_VEL
LIN {X 0,Y 458.386,Z 515.764,A -85,B 0,C 180,E1 -8171.631,E2 -8171.631} C_VEL
LIN {X 0,Y 457.867,Z 529.785,A -85,B 0,C 180,E1 -8172.23,E2 -8172.23} C_VEL
LIN {X 0,Y 457.151,Z 543.537,A -85,B 0,C 180,E1 -8173.015,E2 -8173.015} C_VEL
LIN {X 0,Y 456.451,Z 555.783,A -85,B 0,C 180,E1 -8173.909,E2 -8173.909} C_VEL
LIN {X 0,Y 455.715,Z 567.003,A -85,B 0,C 180,E1 -8174.914,E2 -8174.914} C_VEL
LIN {X 0,Y 454.889,Z 578.279,A -85,B 0,C 180,E1 -8176.143,E2 -8176.143} C_VEL
LIN {X 0,Y 454.298,Z 588.346,A -85,B 0,C 180,E1 -8177.491,E2 -8177.491} C_VEL
LIN {X 0,Y 453.706,Z 596.704,A -85,B 0,C 180,E1 -8178.834,E2 -8178.834} C_VEL
LIN {X 0,Y 453.229,Z 604.686,A -85,B 0,C 180,E1 -8180.403,E2 -8180.403} C_VEL
LIN {X 0,Y 452.878,Z 611.115,A -85,B 0,C 180,E1 -8181.97,E2 -8181.97} C_VEL
LIN {X 0,Y 452.653,Z 616.812,A -85,B 0,C 180,E1 -8183.759,E2 -8183.759} C_VEL
LIN {X 0,Y 452.622,Z 619.066,A -85,B 0,C 180,E1 -8184.653,E2 -8184.653} C_VEL
LIN {X 0,Y 452.489,Z 622.481,A -85,B 0,C 180,E1 -8186.437,E2 -8186.437} C_VEL
LIN {X 0,Y 452.436,Z 624.514,A -85,B 0,C 180,E1 -8188.218,E2 -8188.218} C_VEL
LIN {X 0,Y 452.406,Z 625.216,A -85,B 0,C 180,E1 -8189.999,E2 -8189.999} C_VEL
LIN {X 0,Y 452.434,Z 624.595,A -85,B 0,C 180,E1 -8191.779,E2 -8191.779} C_VEL
LIN {X 0,Y 452.488,Z 622.638,A -85,B 0,C 180,E1 -8193.561,E2 -8193.561} C_VEL
LIN {X 0,Y 452.621,Z 619.293,A -85,B 0,C 180,E1 -8195.344,E2 -8195.344} C_VEL
LIN {X 0,Y 452.752,Z 614.465,A -85,B 0,C 180,E1 -8197.132,E2 -8197.132} C_VEL
LIN {X 0,Y 453.062,Z 608.007,A -85,B 0,C 180,E1 -8198.922,E2 -8198.922} C_VEL
LIN {X 0,Y 453.416,Z 600.817,A -85,B 0,C 180,E1 -8200.492,E2 -8200.492} C_VEL
LIN {X 0,Y 454.068,Z 591.92,A -85,B 0,C 180,E1 -8202.059,E2 -8202.059} C_VEL
LIN {X 0,Y 454.646,Z 582.577,A -85,B 0,C 180,E1 -8203.406,E2 -8203.406} C_VEL
LIN {X 0,Y 455.337,Z 572.225,A -85,B 0,C 180,E1 -8204.638,E2 -8204.638} C_VEL
LIN {X 0,Y 456.09,Z 560.807,A -85,B 0,C 180,E1 -8205.757,E2 -8205.757} C_VEL
LIN {X 0,Y 456.936,Z 548.152,A -85,B 0,C 180,E1 -8206.76,E2 -8206.76} C_VEL
LIN {X 0,Y 457.562,Z 535.848,A -85,B 0,C 180,E1 -8207.541,E2 -8207.541} C_VEL
LIN {X 0,Y 458.229,Z 521.922,A -85,B 0,C 180,E1 -8208.22,E2 -8208.22} C_VEL
LIN {X 0,Y 458.688,Z 507.698,A -85,B 0,C 180,E1 -8208.72,E2 -8208.72} C_VEL
LIN {X 0,Y 459.024,Z 492.886,A -85,B 0,C 180,E1 -8209.043,E2 -8209.043} C_VEL
LIN {X 0,Y 460.27,Z 384.694,A -85,B 0,C 180,E1 -8210.749,E2 -8210.749} C_VEL
LIN {X 0,Y 455.962,Z 363.275,A -85,B 0,C 180,E1 -8211.31,E2 -8211.31} C_VEL
LIN {X 0,Y 456.458,Z 352.194,A -85,B 0,C 180,E1 -8213.356,E2 -8213.356} C_VEL
LIN {X 0,Y 454.136,Z 340.764,A -85,B 0,C 180,E1 -8215.676,E2 -8215.676} C_VEL
LIN {X 0,Y 453.47,Z 337.626,A -85,B 0,C 180,E1 -8216.359,E2 -8216.359} C_VEL
LIN {X 0,Y 453.463,Z 337.626,A -85,B 0,C 180,E1 -8219.782,E2 -8219.782} C_VEL
LIN {X 0,Y 453.477,Z 337.627,A -85,B 0,C 180,E1 -8223.186,E2 -8223.186} C_VEL
LIN {X 0,Y 453.442,Z 337.627,A -85,B 0,C 180,E1 -8226.297,E2 -8226.297} C_VEL
LIN {X 0,Y 453.436,Z 337.627,A -85,B 0,C 180,E1 -8229.453,E2 -8229.453} C_VEL
LIN {X 0,Y 453.427,Z 337.626,A -85,B 0,C 180,E1 -8231.927,E2 -8231.927} C_VEL
LIN {X 0,Y 453.472,Z 337.621,A -85,B 0,C 180,E1 -8235.47,E2 -8235.47} C_VEL
LIN {X 0,Y 453.435,Z 337.626,A -85,B 0,C 180,E1 -8238.204,E2 -8238.204} C_VEL
LIN {X 0,Y 453.437,Z 337.627,A -85,B 0,C 180,E1 -8240.799,E2 -8240.799} C_VEL
LIN {X 0,Y 453.439,Z 337.624,A -85,B 0,C 180,E1 -8243.916,E2 -8243.916} C_VEL
LIN {X 0,Y 453.46,Z 337.616,A -85,B 0,C 180,E1 -8247.149,E2 -8247.149} C_VEL
LIN {X 0,Y 453.448,Z 337.625,A -85,B 0,C 180,E1 -8250.266,E2 -8250.266} C_VEL
LIN {X 0,Y 453.426,Z 337.616,A -85,B 0,C 180,E1 -8253.289,E2 -8253.289} C_VEL
LIN {X 0,Y 453.478,Z 337.62,A -85,B 0,C 180,E1 -8256.237,E2 -8256.237} C_VEL
LIN {X 0,Y 453.467,Z 337.616,A -85,B 0,C 180,E1 -8259.117,E2 -8259.117} C_VEL
LIN {X 0,Y 453.484,Z 337.61,A -85,B 0,C 180,E1 -8261.943,E2 -8261.943} C_VEL
LIN {X 0,Y 453.514,Z 337.621,A -85,B 0,C 180,E1 -8264.725,E2 -8264.725} C_VEL
LIN {X 0,Y 453.541,Z 337.614,A -85,B 0,C 180,E1 -8268.378,E2 -8268.378} C_VEL
LIN {X 0,Y 453.566,Z 337.608,A -85,B 0,C 180,E1 -8271.086,E2 -8271.086} C_VEL
LIN {X 0,Y 453.612,Z 337.602,A -85,B 0,C 180,E1 -8273.774,E2 -8273.774} C_VEL
LIN {X 0,Y 453.698,Z 337.592,A -85,B 0,C 180,E1 -8277.336,E2 -8277.336} C_VEL
LIN {X 0,Y 453.73,Z 337.586,A -85,B 0,C 180,E1 -8280,E2 -8280} C_VEL
LIN {X 0,Y 453.693,Z 337.597,A -85,B 0,C 180,E1 -8282.664,E2 -8282.664} C_VEL
LIN {X 0,Y 453.625,Z 337.604,A -85,B 0,C 180,E1 -8286.226,E2 -8286.226} C_VEL
LIN {X 0,Y 453.542,Z 337.612,A -85,B 0,C 180,E1 -8288.914,E2 -8288.914} C_VEL
LIN {X 0,Y 453.549,Z 337.613,A -85,B 0,C 180,E1 -8292.529,E2 -8292.529} C_VEL
LIN {X 0,Y 453.529,Z 337.617,A -85,B 0,C 180,E1 -8296.196,E2 -8296.196} C_VEL
LIN {X 0,Y 453.502,Z 337.617,A -85,B 0,C 180,E1 -8299.04,E2 -8299.04} C_VEL
LIN {X 0,Y 453.461,Z 337.615,A -85,B 0,C 180,E1 -8301.837,E2 -8301.837} C_VEL
LIN {X 0,Y 453.453,Z 337.626,A -85,B 0,C 180,E1 -8304.738,E2 -8304.738} C_VEL
LIN {X 0,Y 453.449,Z 337.623,A -85,B 0,C 180,E1 -8307.944,E2 -8307.944} C_VEL
LIN {X 0,Y 453.443,Z 337.626,A -85,B 0,C 180,E1 -8310.762,E2 -8310.762} C_VEL
LIN {X 0,Y 453.452,Z 337.623,A -85,B 0,C 180,E1 -8313.915,E2 -8313.915} C_VEL
LIN {X 0,Y 453.422,Z 337.627,A -85,B 0,C 180,E1 -8317.193,E2 -8317.193} C_VEL
LIN {X 0,Y 453.454,Z 337.625,A -85,B 0,C 180,E1 -8320.613,E2 -8320.613} C_VEL
LIN {X 0,Y 453.469,Z 337.626,A -85,B 0,C 180,E1 -8324.529,E2 -8324.529} C_VEL
LIN {X 0,Y 453.42,Z 337.634,A -85,B 0,C 180,E1 -8328.073,E2 -8328.073} C_VEL
LIN {X 0,Y 453.414,Z 337.631,A -85,B 0,C 180,E1 -8330.806,E2 -8330.806} C_VEL
LIN {X 0,Y 453.432,Z 337.632,A -85,B 0,C 180,E1 -8333.917,E2 -8333.917} C_VEL
LIN {X 0,Y 453.464,Z 337.623,A -85,B 0,C 180,E1 -8337.152,E2 -8337.152} C_VEL
LIN {X 0,Y 453.454,Z 337.624,A -85,B 0,C 180,E1 -8340.269,E2 -8340.269} C_VEL
LIN {X 0,Y 453.494,Z 337.642,A -85,B 0,C 180,E1 -8342.547,E2 -8342.547} C_VEL
LIN {X 0,Y 456.649,Z 352.459,A -85,B 0,C 180,E1 -8345.448,E2 -8345.448} C_VEL
LIN {X 0,Y 456.735,Z 356.493,A -85,B 0,C 180,E1 -8346.178,E2 -8346.178} C_VEL
LIN {X 0,Y 455.888,Z 371.028,A -85,B 0,C 180,E1 -8348.724,E2 -8348.724} C_VEL
LIN {X 0,Y 460.162,Z 393.864,A -85,B 0,C 180,E1 -8349.308,E2 -8349.308} C_VEL
LIN {X 0,Y 458.859,Z 507.891,A -85,B 0,C 180,E1 -8351.124,E2 -8351.124} C_VEL
LIN {X 0,Y 458.394,Z 522.043,A -85,B 0,C 180,E1 -8351.509,E2 -8351.509} C_VEL
LIN {X 0,Y 457.833,Z 535.749,A -85,B 0,C 180,E1 -8352.065,E2 -8352.065} C_VEL
LIN {X 0,Y 457.234,Z 548.596,A -85,B 0,C 180,E1 -8352.761,E2 -8352.761} C_VEL
LIN {X 0,Y 456.471,Z 561.862,A -85,B 0,C 180,E1 -8353.683,E2 -8353.683} C_VEL
LIN {X 0,Y 455.646,Z 573.499,A -85,B 0,C 180,E1 -8354.686,E2 -8354.686} C_VEL
LIN {X 0,Y 454.847,Z 585.141,A -85,B 0,C 180,E1 -8355.917,E2 -8355.917} C_VEL
LIN {X 0,Y 454.197,Z 595.666,A -85,B 0,C 180,E1 -8357.279,E2 -8357.279} C_VEL
LIN {X 0,Y 453.698,Z 604.141,A -85,B 0,C 180,E1 -8358.61,E2 -8358.61} C_VEL
LIN {X 0,Y 453.179,Z 612.365,A -85,B 0,C 180,E1 -8360.179,E2 -8360.179} C_VEL
LIN {X 0,Y 452.888,Z 618.119,A -85,B 0,C 180,E1 -8361.524,E2 -8361.524} C_VEL
LIN {X 0,Y 452.663,Z 622.834,A -85,B 0,C 180,E1 -8362.866,E2 -8362.866} C_VEL
LIN {X 0,Y 452.591,Z 627.725,A -85,B 0,C 180,E1 -8364.655,E2 -8364.655} C_VEL
LIN {X 0,Y 452.446,Z 631.122,A -85,B 0,C 180,E1 -8366.439,E2 -8366.439} C_VEL
LIN {X 0,Y 452.429,Z 633.128,A -85,B 0,C 180,E1 -8368.221,E2 -8368.221} C_VEL
LIN {X 0,Y 452.405,Z 633.791,A -85,B 0,C 180,E1 -8370.001,E2 -8370.001} C_VEL
LIN {X 0,Y 452.43,Z 633.123,A -85,B 0,C 180,E1 -8371.782,E2 -8371.782} C_VEL
LIN {X 0,Y 452.446,Z 631.111,A -85,B 0,C 180,E1 -8373.564,E2 -8373.564} C_VEL
LIN {X 0,Y 452.586,Z 627.712,A -85,B 0,C 180,E1 -8375.347,E2 -8375.347} C_VEL
LIN {X 0,Y 452.663,Z 622.823,A -85,B 0,C 180,E1 -8377.136,E2 -8377.136} C_VEL
LIN {X 0,Y 452.967,Z 616.29,A -85,B 0,C 180,E1 -8378.927,E2 -8378.927} C_VEL
LIN {X 0,Y 453.338,Z 609.019,A -85,B 0,C 180,E1 -8380.497,E2 -8380.497} C_VEL
LIN {X 0,Y 453.988,Z 600.018,A -85,B 0,C 180,E1 -8382.064,E2 -8382.064} C_VEL
LIN {X 0,Y 454.503,Z 590.567,A -85,B 0,C 180,E1 -8383.413,E2 -8383.413} C_VEL
LIN {X 0,Y 455.225,Z 580.108,A -85,B 0,C 180,E1 -8384.645,E2 -8384.645} C_VEL
LIN {X 0,Y 456.005,Z 568.561,A -85,B 0,C 180,E1 -8385.763,E2 -8385.763} C_VEL
LIN {X 0,Y 456.826,Z 555.75,A -85,B 0,C 180,E1 -8386.767,E2 -8386.767} C_VEL
LIN {X 0,Y 457.592,Z 542.589,A -85,B 0,C 180,E1 -8387.582,E2 -8387.582} C_VEL
LIN {X 0,Y 458.112,Z 529.323,A -85,B 0,C 180,E1 -8388.216,E2 -8388.216} C_VEL
LIN {X 0,Y 458.675,Z 515.581,A -85,B 0,C 180,E1 -8388.684,E2 -8388.684} C_VEL
LIN {X 0,Y 458.945,Z 501.572,A -85,B 0,C 180,E1 -8388.992,E2 -8388.992} C_VEL
LIN {X 0,Y 460.103,Z 393.201,A -85,B 0,C 180,E1 -8390.703,E2 -8390.703} C_VEL
LIN {X 0,Y 455.879,Z 370.971,A -85,B 0,C 180,E1 -8391.283,E2 -8391.283} C_VEL
LIN {X 0,Y 456.831,Z 355.11,A -85,B 0,C 180,E1 -8394.06,E2 -8394.06} C_VEL
LIN {X 0,Y 456.107,Z 349.726,A -85,B 0,C 180,E1 -8395.071,E2 -8395.071} C_VEL
LIN {X 0,Y 453.504,Z 337.623,A -85,B 0,C 180,E1 -8397.455,E2 -8397.455} C_VEL
LIN {X 0,Y 453.478,Z 337.623,A -85,B 0,C 180,E1 -8400.761,E2 -8400.761} C_VEL
LIN {X 0,Y 453.481,Z 337.622,A -85,B 0,C 180,E1 -8403.913,E2 -8403.913} C_VEL
LIN {X 0,Y 453.454,Z 337.626,A -85,B 0,C 180,E1 -8407.191,E2 -8407.191} C_VEL
LIN {X 0,Y 453.491,Z 337.621,A -85,B 0,C 180,E1 -8409.451,E2 -8409.451} C_VEL
LIN {X 0,Y 453.481,Z 337.619,A -85,B 0,C 180,E1 -8411.935,E2 -8411.935} C_VEL
LIN {X 0,Y 453.492,Z 337.62,A -85,B 0,C 180,E1 -8415.471,E2 -8415.471} C_VEL
LIN {X 0,Y 453.484,Z 337.621,A -85,B 0,C 180,E1 -8418.21,E2 -8418.21} C_VEL
LIN {X 0,Y 453.514,Z 337.62,A -85,B 0,C 180,E1 -8420.792,E2 -8420.792} C_VEL
LIN {X 0,Y 453.456,Z 337.624,A -85,B 0,C 180,E1 -8423.917,E2 -8423.917} C_VEL
LIN {X 0,Y 453.488,Z 337.622,A -85,B 0,C 180,E1 -8427.152,E2 -8427.152} C_VEL
LIN {X 0,Y 453.472,Z 337.629,A -85,B 0,C 180,E1 -8430.268,E2 -8430.268} C_VEL
LIN {X 0,Y 453.467,Z 337.63,A -85,B 0,C 180,E1 -8433.291,E2 -8433.291} C_VEL
LIN {X 0,Y 453.509,Z 337.686,A -85,B 0,C 180,E1 -8435.315,E2 -8435.315} C_VEL
LIN {X 0,Y 455.642,Z 347.225,A -85,B 0,C 180,E1 -8437.079,E2 -8437.079} C_VEL
LIN {X 0,Y 456.133,Z 351.257,A -85,B 0,C 180,E1 -8437.8,E2 -8437.8} C_VEL
LIN {X 0,Y 455.713,Z 369.476,A -85,B 0,C 180,E1 -8440.893,E2 -8440.893} C_VEL
LIN {X 0,Y 455.515,Z 378.124,A -85,B 0,C 180,E1 -8442.356,E2 -8442.356} C_VEL
LIN {X 0,Y 458.148,Z 391.623,A -85,B 0,C 180,E1 -8442.773,E2 -8442.773} C_VEL
LIN {X 0,Y 456.567,Z 487.579,A -85,B 0,C 180,E1 -8444.63,E2 -8444.63} C_VEL
LIN {X 0,Y 456.257,Z 500.369,A -85,B 0,C 180,E1 -8445.048,E2 -8445.048} C_VEL
LIN {X 0,Y 455.854,Z 513.33,A -85,B 0,C 180,E1 -8445.662,E2 -8445.662} C_VEL
LIN {X 0,Y 455.403,Z 525.178,A -85,B 0,C 180,E1 -8446.411,E2 -8446.411} C_VEL
LIN {X 0,Y 454.928,Z 537.366,A -85,B 0,C 180,E1 -8447.411,E2 -8447.411} C_VEL
LIN {X 0,Y 454.385,Z 547.085,A -85,B 0,C 180,E1 -8448.4,E2 -8448.4} C_VEL
LIN {X 0,Y 453.951,Z 555.99,A -85,B 0,C 180,E1 -8449.519,E2 -8449.519} C_VEL
LIN {X 0,Y 453.504,Z 564.67,A -85,B 0,C 180,E1 -8450.86,E2 -8450.86} C_VEL
LIN {X 0,Y 453.166,Z 571.598,A -85,B 0,C 180,E1 -8452.201,E2 -8452.201} C_VEL
LIN {X 0,Y 452.966,Z 577.892,A -85,B 0,C 180,E1 -8453.765,E2 -8453.765} C_VEL
LIN {X 0,Y 452.683,Z 581.993,A -85,B 0,C 180,E1 -8455.102,E2 -8455.102} C_VEL
LIN {X 0,Y 452.692,Z 584.993,A -85,B 0,C 180,E1 -8456.44,E2 -8456.44} C_VEL
LIN {X 0,Y 452.593,Z 586.45,A -85,B 0,C 180,E1 -8457.33,E2 -8457.33} C_VEL
LIN {X 0,Y 452.546,Z 587.446,A -85,B 0,C 180,E1 -8458.22,E2 -8458.22} C_VEL
LIN {X 0,Y 452.492,Z 588.046,A -85,B 0,C 180,E1 -8459.11,E2 -8459.11} C_VEL
LIN {X 0,Y 452.469,Z 588.241,A -85,B 0,C 180,E1 -8460,E2 -8460} C_VEL
LIN {X 0,Y 452.492,Z 587.977,A -85,B 0,C 180,E1 -8460.89,E2 -8460.89} C_VEL
LIN {X 0,Y 452.517,Z 587.312,A -85,B 0,C 180,E1 -8461.78,E2 -8461.78} C_VEL
LIN {X 0,Y 452.577,Z 586.248,A -85,B 0,C 180,E1 -8462.67,E2 -8462.67} C_VEL
LIN {X 0,Y 452.668,Z 584.727,A -85,B 0,C 180,E1 -8463.561,E2 -8463.561} C_VEL
LIN {X 0,Y 452.634,Z 581.624,A -85,B 0,C 180,E1 -8464.899,E2 -8464.899} C_VEL
LIN {X 0,Y 452.895,Z 577.424,A -85,B 0,C 180,E1 -8466.236,E2 -8466.236} C_VEL
LIN {X 0,Y 453.042,Z 571.01,A -85,B 0,C 180,E1 -8467.801,E2 -8467.801} C_VEL
LIN {X 0,Y 453.395,Z 563.962,A -85,B 0,C 180,E1 -8469.142,E2 -8469.142} C_VEL
LIN {X 0,Y 453.812,Z 555.146,A -85,B 0,C 180,E1 -8470.484,E2 -8470.484} C_VEL
LIN {X 0,Y 454.23,Z 546.113,A -85,B 0,C 180,E1 -8471.604,E2 -8471.604} C_VEL
LIN {X 0,Y 454.734,Z 535.495,A -85,B 0,C 180,E1 -8472.665,E2 -8472.665} C_VEL
LIN {X 0,Y 455.178,Z 523.578,A -85,B 0,C 180,E1 -8473.619,E2 -8473.619} C_VEL
LIN {X 0,Y 455.634,Z 510.735,A -85,B 0,C 180,E1 -8474.402,E2 -8474.402} C_VEL
LIN {X 0,Y 456.012,Z 498.504,A -85,B 0,C 180,E1 -8474.96,E2 -8474.96} C_VEL
LIN {X 0,Y 456.376,Z 484.976,A -85,B 0,C 180,E1 -8475.377,E2 -8475.377} C_VEL
LIN {X 0,Y 457.415,Z 390.713,A -85,B 0,C 180,E1 -8477.08,E2 -8477.08} C_VEL
LIN {X 0,Y 454.819,Z 376.054,A -85,B 0,C 180,E1 -8477.451,E2 -8477.451} C_VEL
LIN {X 0,Y 455.315,Z 358.384,A -85,B 0,C 180,E1 -8480.558,E2 -8480.558} C_VEL
LIN {X 0,Y 455.468,Z 347.997,A -85,B 0,C 180,E1 -8482.39,E2 -8482.39} C_VEL
LIN {X 0,Y 453.549,Z 337.617,A -85,B 0,C 180,E1 -8484.355,E2 -8484.355} C_VEL
LIN {X 0,Y 453.537,Z 337.618,A -85,B 0,C 180,E1 -8487.959,E2 -8487.959} C_VEL
LIN {X 0,Y 453.471,Z 337.62,A -85,B 0,C 180,E1 -8491.525,E2 -8491.525} C_VEL
LIN {X 0,Y 453.492,Z 337.618,A -85,B 0,C 180,E1 -8494.777,E2 -8494.777} C_VEL
LIN {X 0,Y 453.462,Z 337.624,A -85,B 0,C 180,E1 -8498.312,E2 -8498.312} C_VEL
LIN {X 0,Y 453.476,Z 337.62,A -85,B 0,C 180,E1 -8500.611,E2 -8500.611} C_VEL
LIN {X 0,Y 453.466,Z 337.624,A -85,B 0,C 180,E1 -8504.221,E2 -8504.221} C_VEL
LIN {X 0,Y 453.442,Z 337.626,A -85,B 0,C 180,E1 -8507.001,E2 -8507.001} C_VEL
LIN {X 0,Y 453.476,Z 337.625,A -85,B 0,C 180,E1 -8509.412,E2 -8509.412} C_VEL
LIN {X 0,Y 453.444,Z 337.626,A -85,B 0,C 180,E1 -8512.808,E2 -8512.808} C_VEL
LIN {X 0,Y 453.467,Z 337.624,A -85,B 0,C 180,E1 -8516.085,E2 -8516.085} C_VEL
LIN {X 0,Y 453.457,Z 337.627,A -85,B 0,C 180,E1 -8519.238,E2 -8519.238} C_VEL
LIN {X 0,Y 453.475,Z 337.623,A -85,B 0,C 180,E1 -8522.292,E2 -8522.292} C_VEL
LIN {X 0,Y 453.484,Z 337.778,A -85,B 0,C 180,E1 -8523.798,E2 -8523.798} C_VEL
LIN {X 0,Y 456.394,Z 351.679,A -85,B 0,C 180,E1 -8526.638,E2 -8526.638} C_VEL
LIN {X 0,Y 456.526,Z 354.344,A -85,B 0,C 180,E1 -8527.147,E2 -8527.147} C_VEL
LIN {X 0,Y 455.734,Z 356.856,A -85,B 0,C 180,E1 -8527.552,E2 -8527.552} C_VEL
LIN {X 0,Y 452.997,Z 361.616,A -85,B 0,C 180,E1 -8528.105,E2 -8528.105} C_VEL
LIN {X 0,Y 451.056,Z 366.007,A -85,B 0,C 180,E1 -8528.436,E2 -8528.436} C_VEL
LIN {X 0,Y 450.554,Z 369.719,A -85,B 0,C 180,E1 -8528.613,E2 -8528.613} C_VEL
LIN {X 0,Y 450.701,Z 371.004,A -85,B 0,C 180,E1 -8528.654,E2 -8528.654} C_VEL
LIN {X 0,Y 453.591,Z 385.869,A -85,B 0,C 180,E1 -8529.044,E2 -8529.044} C_VEL
LIN {X 0,Y 452.203,Z 498.652,A -85,B 0,C 180,E1 -8530.862,E2 -8530.862} C_VEL
LIN {X 0,Y 451.778,Z 513.303,A -85,B 0,C 180,E1 -8531.255,E2 -8531.255} C_VEL
LIN {X 0,Y 451.277,Z 526.815,A -85,B 0,C 180,E1 -8531.803,E2 -8531.803} C_VEL
LIN {X 0,Y 450.619,Z 539.231,A -85,B 0,C 180,E1 -8532.471,E2 -8532.471} C_VEL
LIN {X 0,Y 449.934,Z 551.584,A -85,B 0,C 180,E1 -8533.319,E2 -8533.319} C_VEL
LIN {X 0,Y 449.053,Z 563.559,A -85,B 0,C 180,E1 -8534.336,E2 -8534.336} C_VEL
LIN {X 0,Y 448.246,Z 574.479,A -85,B 0,C 180,E1 -8535.47,E2 -8535.47} C_VEL
LIN {X 0,Y 447.597,Z 583.696,A -85,B 0,C 180,E1 -8536.618,E2 -8536.618} C_VEL
LIN {X 0,Y 447.037,Z 592.785,A -85,B 0,C 180,E1 -8537.976,E2 -8537.976} C_VEL
LIN {X 0,Y 446.389,Z 601.532,A -85,B 0,C 180,E1 -8539.567,E2 -8539.567} C_VEL
LIN {X 0,Y 446.021,Z 607.698,A -85,B 0,C 180,E1 -8540.933,E2 -8540.933} C_VEL
LIN {X 0,Y 445.685,Z 614.237,A -85,B 0,C 180,E1 -8542.751,E2 -8542.751} C_VEL
LIN {X 0,Y 445.541,Z 619.135,A -85,B 0,C 180,E1 -8544.568,E2 -8544.568} C_VEL
LIN {X 0,Y 445.389,Z 622.549,A -85,B 0,C 180,E1 -8546.38,E2 -8546.38} C_VEL
LIN {X 0,Y 445.433,Z 623.733,A -85,B 0,C 180,E1 -8547.286,E2 -8547.286} C_VEL
LIN {X 0,Y 445.313,Z 625.097,A -85,B 0,C 180,E1 -8549.094,E2 -8549.094} C_VEL
LIN {X 0,Y 445.313,Z 625.137,A -85,B 0,C 180,E1 -8550.903,E2 -8550.903} C_VEL
LIN {X 0,Y 445.432,Z 623.852,A -85,B 0,C 180,E1 -8552.712,E2 -8552.712} C_VEL
LIN {X 0,Y 445.424,Z 621.21,A -85,B 0,C 180,E1 -8554.523,E2 -8554.523} C_VEL
LIN {X 0,Y 445.577,Z 617.139,A -85,B 0,C 180,E1 -8556.337,E2 -8556.337} C_VEL
LIN {X 0,Y 445.826,Z 611.517,A -85,B 0,C 180,E1 -8558.155,E2 -8558.155} C_VEL
LIN {X 0,Y 446.191,Z 605.173,A -85,B 0,C 180,E1 -8559.747,E2 -8559.747} C_VEL
LIN {X 0,Y 446.698,Z 597.283,A -85,B 0,C 180,E1 -8561.341,E2 -8561.341} C_VEL
LIN {X 0,Y 447.239,Z 589.029,A -85,B 0,C 180,E1 -8562.707,E2 -8562.707} C_VEL
LIN {X 0,Y 447.922,Z 579.085,A -85,B 0,C 180,E1 -8564.074,E2 -8564.074} C_VEL
LIN {X 0,Y 448.757,Z 568.015,A -85,B 0,C 180,E1 -8565.323,E2 -8565.323} C_VEL
LIN {X 0,Y 449.529,Z 556.999,A -85,B 0,C 180,E1 -8566.343,E2 -8566.343} C_VEL
LIN {X 0,Y 450.305,Z 545.042,A -85,B 0,C 180,E1 -8567.248,E2 -8567.248} C_VEL
LIN {X 0,Y 451.02,Z 531.844,A -85,B 0,C 180,E1 -8568.038,E2 -8568.038} C_VEL
LIN {X 0,Y 451.623,Z 518.089,A -85,B 0,C 180,E1 -8568.66,E2 -8568.66} C_VEL
LIN {X 0,Y 452.093,Z 503.843,A -85,B 0,C 180,E1 -8569.111,E2 -8569.111} C_VEL
LIN {X 0,Y 452.441,Z 483.983,A -85,B 0,C 180,E1 -8569.479,E2 -8569.479} C_VEL
LIN {X 0,Y 453.556,Z 384.805,A -85,B 0,C 180,E1 -8571.069,E2 -8571.069} C_VEL
LIN {X 0,Y 449.13,Z 363.229,A -85,B 0,C 180,E1 -8571.671,E2 -8571.671} C_VEL
LIN {X 0,Y 449.677,Z 354.799,A -85,B 0,C 180,E1 -8573.241,E2 -8573.241} C_VEL
LIN {X 0,Y 448.011,Z 345.906,A -85,B 0,C 180,E1 -8575.057,E2 -8575.057} C_VEL
LIN {X 0,Y 446.42,Z 338.505,A -85,B 0,C 180,E1 -8576.656,E2 -8576.656} C_VEL
LIN {X 0,Y 446.42,Z 338.503,A -85,B 0,C 180,E1 -8580.018,E2 -8580.018} C_VEL
LIN {X 0,Y 446.439,Z 338.502,A -85,B 0,C 180,E1 -8583.452,E2 -8583.452} C_VEL
LIN {X 0,Y 446.391,Z 338.508,A -85,B 0,C 180,E1 -8586.744,E2 -8586.744} C_VEL
LIN {X 0,Y 446.389,Z 338.504,A -85,B 0,C 180,E1 -8589.514,E2 -8589.514} C_VEL
LIN {X 0,Y 446.366,Z 338.51,A -85,B 0,C 180,E1 -8592.61,E2 -8592.61} C_VEL
LIN {X 0,Y 446.44,Z 338.501,A -85,B 0,C 180,E1 -8595.103,E2 -8595.103} C_VEL
LIN {X 0,Y 446.391,Z 338.507,A -85,B 0,C 180,E1 -8598.605,E2 -8598.605} C_VEL
LIN {X 0,Y 446.399,Z 338.495,A -85,B 0,C 180,E1 -8601.92,E2 -8601.92} C_VEL
LIN {X 0,Y 446.409,Z 338.499,A -85,B 0,C 180,E1 -8605.475,E2 -8605.475} C_VEL
LIN {X 0,Y 446.397,Z 338.501,A -85,B 0,C 180,E1 -8608.698,E2 -8608.698} C_VEL
LIN {X 0,Y 446.41,Z 338.497,A -85,B 0,C 180,E1 -8611.835,E2 -8611.835} C_VEL
LIN {X 0,Y 446.415,Z 338.497,A -85,B 0,C 180,E1 -8614.845,E2 -8614.845} C_VEL
LIN {X 0,Y 446.434,Z 338.499,A -85,B 0,C 180,E1 -8618.244,E2 -8618.244} C_VEL
LIN {X 0,Y 446.434,Z 338.487,A -85,B 0,C 180,E1 -8621.648,E2 -8621.648} C_VEL
LIN {X 0,Y 446.477,Z 338.496,A -85,B 0,C 180,E1 -8624.479,E2 -8624.479} C_VEL
LIN {X 0,Y 446.5,Z 338.489,A -85,B 0,C 180,E1 -8628.192,E2 -8628.192} C_VEL
LIN {X 0,Y 446.514,Z 338.488,A -85,B 0,C 180,E1 -8630.944,E2 -8630.944} C_VEL
LIN {X 0,Y 446.583,Z 338.478,A -85,B 0,C 180,E1 -8633.675,E2 -8633.675} C_VEL
LIN {X 0,Y 446.647,Z 338.471,A -85,B 0,C 180,E1 -8637.294,E2 -8637.294} C_VEL
LIN {X 0,Y 446.681,Z 338.464,A -85,B 0,C 180,E1 -8640,E2 -8640} C_VEL
LIN {X 0,Y 446.642,Z 338.474,A -85,B 0,C 180,E1 -8642.706,E2 -8642.706} C_VEL
LIN {X 0,Y 446.594,Z 338.481,A -85,B 0,C 180,E1 -8646.324,E2 -8646.324} C_VEL
LIN {X 0,Y 446.493,Z 338.489,A -85,B 0,C 180,E1 -8649.056,E2 -8649.056} C_VEL
LIN {X 0,Y 446.507,Z 338.489,A -85,B 0,C 180,E1 -8652.73,E2 -8652.73} C_VEL
LIN {X 0,Y 446.473,Z 338.495,A -85,B 0,C 180,E1 -8656.46,E2 -8656.46} C_VEL
LIN {X 0,Y 446.453,Z 338.494,A -85,B 0,C 180,E1 -8659.304,E2 -8659.304} C_VEL
LIN {X 0,Y 446.402,Z 338.494,A -85,B 0,C 180,E1 -8662.2,E2 -8662.2} C_VEL
LIN {X 0,Y 446.405,Z 338.501,A -85,B 0,C 180,E1 -8665.155,E2 -8665.155} C_VEL
LIN {X 0,Y 446.423,Z 338.496,A -85,B 0,C 180,E1 -8668.183,E2 -8668.183} C_VEL
LIN {X 0,Y 446.394,Z 338.502,A -85,B 0,C 180,E1 -8671.302,E2 -8671.302} C_VEL
LIN {X 0,Y 446.407,Z 338.505,A -85,B 0,C 180,E1 -8674.525,E2 -8674.525} C_VEL
LIN {X 0,Y 446.382,Z 338.509,A -85,B 0,C 180,E1 -8678.077,E2 -8678.077} C_VEL
LIN {X 0,Y 446.383,Z 338.502,A -85,B 0,C 180,E1 -8681.396,E2 -8681.396} C_VEL
LIN {X 0,Y 446.409,Z 338.501,A -85,B 0,C 180,E1 -8685.109,E2 -8685.109} C_VEL
LIN {X 0,Y 446.384,Z 338.508,A -85,B 0,C 180,E1 -8688.606,E2 -8688.606} C_VEL
LIN {X 0,Y 446.379,Z 338.511,A -85,B 0,C 180,E1 -8692.12,E2 -8692.12} C_VEL
LIN {X 0,Y 446.411,Z 338.503,A -85,B 0,C 180,E1 -8695.478,E2 -8695.478} C_VEL
LIN {X 0,Y 446.4,Z 338.504,A -85,B 0,C 180,E1 -8698.7,E2 -8698.7} C_VEL
LIN {X 0,Y 446.421,Z 338.504,A -85,B 0,C 180,E1 -8702.084,E2 -8702.084} C_VEL
LIN {X 0,Y 446.455,Z 338.602,A -85,B 0,C 180,E1 -8702.27,E2 -8702.27} C_VEL
LIN {X 0,Y 449.679,Z 353.487,A -85,B 0,C 180,E1 -8705.242,E2 -8705.242} C_VEL
LIN {X 0,Y 449.851,Z 357.775,A -85,B 0,C 180,E1 -8706.036,E2 -8706.036} C_VEL
LIN {X 0,Y 449.048,Z 370.977,A -85,B 0,C 180,E1 -8708.386,E2 -8708.386} C_VEL
LIN {X 0,Y 453.513,Z 394.417,A -85,B 0,C 180,E1 -8709,E2 -8709} C_VEL
LIN {X 0,Y 452.143,Z 507.838,A -85,B 0,C 180,E1 -8710.832,E2 -8710.832} C_VEL
LIN {X 0,Y 451.679,Z 521.984,A -85,B 0,C 180,E1 -8711.224,E2 -8711.224} C_VEL
LIN {X 0,Y 451.096,Z 535.688,A -85,B 0,C 180,E1 -8711.787,E2 -8711.787} C_VEL
LIN {X 0,Y 450.421,Z 548.805,A -85,B 0,C 180,E1 -8712.51,E2 -8712.51} C_VEL
LIN {X 0,Y 449.641,Z 561.798,A -85,B 0,C 180,E1 -8713.428,E2 -8713.428} C_VEL
LIN {X 0,Y 448.772,Z 573.434,A -85,B 0,C 180,E1 -8714.445,E2 -8714.445} C_VEL
LIN {X 0,Y 447.943,Z 585.076,A -85,B 0,C 180,E1 -8715.695,E2 -8715.695} C_VEL
LIN {X 0,Y 447.294,Z 594.666,A -85,B 0,C 180,E1 -8716.947,E2 -8716.947} C_VEL
LIN {X 0,Y 446.695,Z 604.075,A -85,B 0,C 180,E1 -8718.429,E2 -8718.429} C_VEL
LIN {X 0,Y 446.125,Z 612.298,A -85,B 0,C 180,E1 -8720.022,E2 -8720.022} C_VEL
LIN {X 0,Y 445.824,Z 618.052,A -85,B 0,C 180,E1 -8721.389,E2 -8721.389} C_VEL
LIN {X 0,Y 445.589,Z 622.767,A -85,B 0,C 180,E1 -8722.753,E2 -8722.753} C_VEL
LIN {X 0,Y 445.507,Z 627.658,A -85,B 0,C 180,E1 -8724.57,E2 -8724.57} C_VEL
LIN {X 0,Y 445.345,Z 631.055,A -85,B 0,C 180,E1 -8726.382,E2 -8726.382} C_VEL
LIN {X 0,Y 445.349,Z 633.061,A -85,B 0,C 180,E1 -8728.193,E2 -8728.193} C_VEL
LIN {X 0,Y 445.314,Z 633.724,A -85,B 0,C 180,E1 -8730.001,E2 -8730.001} C_VEL
LIN {X 0,Y 445.349,Z 633.055,A -85,B 0,C 180,E1 -8731.81,E2 -8731.81} C_VEL
LIN {X 0,Y 445.346,Z 631.043,A -85,B 0,C 180,E1 -8733.62,E2 -8733.62} C_VEL
LIN {X 0,Y 445.498,Z 627.644,A -85,B 0,C 180,E1 -8735.433,E2 -8735.433} C_VEL
LIN {X 0,Y 445.59,Z 622.754,A -85,B 0,C 180,E1 -8737.25,E2 -8737.25} C_VEL
LIN {X 0,Y 445.923,Z 616.221,A -85,B 0,C 180,E1 -8739.069,E2 -8739.069} C_VEL
LIN {X 0,Y 446.33,Z 608.95,A -85,B 0,C 180,E1 -8740.663,E2 -8740.663} C_VEL
LIN {X 0,Y 446.999,Z 599.949,A -85,B 0,C 180,E1 -8742.256,E2 -8742.256} C_VEL
LIN {X 0,Y 447.553,Z 590.497,A -85,B 0,C 180,E1 -8743.625,E2 -8743.625} C_VEL
LIN {X 0,Y 448.326,Z 580.037,A -85,B 0,C 180,E1 -8744.875,E2 -8744.875} C_VEL
LIN {X 0,Y 449.157,Z 568.49,A -85,B 0,C 180,E1 -8746.01,E2 -8746.01} C_VEL
LIN {X 0,Y 450.011,Z 555.678,A -85,B 0,C 180,E1 -8747.028,E2 -8747.028} C_VEL
LIN {X 0,Y 450.806,Z 542.357,A -85,B 0,C 180,E1 -8747.865,E2 -8747.865} C_VEL
LIN {X 0,Y 451.375,Z 529.249,A -85,B 0,C 180,E1 -8748.497,E2 -8748.497} C_VEL
LIN {X 0,Y 451.969,Z 515.505,A -85,B 0,C 180,E1 -8748.972,E2 -8748.972} C_VEL
LIN {X 0,Y 452.236,Z 501.488,A -85,B 0,C 180,E1 -8749.284,E2 -8749.284} C_VEL
LIN {X 0,Y 453.515,Z 394.601,A -85,B 0,C 180,E1 -8750.993,E2 -8750.993} C_VEL
LIN {X 0,Y 449.044,Z 370.951,A -85,B 0,C 180,E1 -8751.615,E2 -8751.615} C_VEL
LIN {X 0,Y 449.954,Z 356.397,A -85,B 0,C 180,E1 -8754.205,E2 -8754.205} C_VEL
LIN {X 0,Y 448.875,Z 349.655,A -85,B 0,C 180,E1 -8755.505,E2 -8755.505} C_VEL
LIN {X 0,Y 446.441,Z 338.502,A -85,B 0,C 180,E1 -8757.764,E2 -8757.764} C_VEL
LIN {X 0,Y 446.429,Z 338.501,A -85,B 0,C 180,E1 -8760.251,E2 -8760.251} C_VEL
LIN {X 0,Y 446.45,Z 338.5,A -85,B 0,C 180,E1 -8763.454,E2 -8763.454} C_VEL
LIN {X 0,Y 446.405,Z 338.502,A -85,B 0,C 180,E1 -8766.746,E2 -8766.746} C_VEL
LIN {X 0,Y 446.447,Z 338.495,A -85,B 0,C 180,E1 -8770.199,E2 -8770.199} C_VEL
LIN {X 0,Y 446.434,Z 338.499,A -85,B 0,C 180,E1 -8772.605,E2 -8772.605} C_VEL
LIN {X 0,Y 446.459,Z 338.5,A -85,B 0,C 180,E1 -8775.104,E2 -8775.104} C_VEL
LIN {X 0,Y 446.433,Z 338.5,A -85,B 0,C 180,E1 -8778.61,E2 -8778.61} C_VEL
LIN {X 0,Y 446.46,Z 338.497,A -85,B 0,C 180,E1 -8780.975,E2 -8780.975} C_VEL
LIN {X 0,Y 446.422,Z 338.505,A -85,B 0,C 180,E1 -8784.374,E2 -8784.374} C_VEL
LIN {X 0,Y 446.427,Z 338.503,A -85,B 0,C 180,E1 -8787.639,E2 -8787.639} C_VEL
LIN {X 0,Y 446.442,Z 338.505,A -85,B 0,C 180,E1 -8790.79,E2 -8790.79} C_VEL
LIN {X 0,Y 446.44,Z 338.505,A -85,B 0,C 180,E1 -8793.846,E2 -8793.846} C_VEL
LIN {X 0,Y 446.492,Z 338.699,A -85,B 0,C 180,E1 -8794.972,E2 -8794.972} C_VEL
LIN {X 0,Y 448.898,Z 349.204,A -85,B 0,C 180,E1 -8796.958,E2 -8796.958} C_VEL
LIN {X 0,Y 449.33,Z 353.652,A -85,B 0,C 180,E1 -8797.765,E2 -8797.765} C_VEL
LIN {X 0,Y 448.937,Z 370.312,A -85,B 0,C 180,E1 -8800.613,E2 -8800.613} C_VEL
LIN {X 0,Y 448.701,Z 378.446,A -85,B 0,C 180,E1 -8802.006,E2 -8802.006} C_VEL
LIN {X 0,Y 451.449,Z 392.188,A -85,B 0,C 180,E1 -8802.454,E2 -8802.454} C_VEL
LIN {X 0,Y 449.93,Z 478.647,A -85,B 0,C 180,E1 -8804.165,E2 -8804.165} C_VEL
LIN {X 0,Y 449.716,Z 492.555,A -85,B 0,C 180,E1 -8804.506,E2 -8804.506} C_VEL
LIN {X 0,Y 449.34,Z 505.153,A -85,B 0,C 180,E1 -8804.986,E2 -8804.986} C_VEL
LIN {X 0,Y 448.972,Z 516.876,A -85,B 0,C 180,E1 -8805.611,E2 -8805.611} C_VEL
LIN {X 0,Y 448.398,Z 528.429,A -85,B 0,C 180,E1 -8806.402,E2 -8806.402} C_VEL
LIN {X 0,Y 447.971,Z 538.944,A -85,B 0,C 180,E1 -8807.312,E2 -8807.312} C_VEL
LIN {X 0,Y 447.361,Z 549.467,A -85,B 0,C 180,E1 -8808.445,E2 -8808.445} C_VEL
LIN {X 0,Y 446.918,Z 558.039,A -85,B 0,C 180,E1 -8809.581,E2 -8809.581} C_VEL
LIN {X 0,Y 446.445,Z 566.358,A -85,B 0,C 180,E1 -8810.943,E2 -8810.943} C_VEL
LIN {X 0,Y 446.088,Z 573.019,A -85,B 0,C 180,E1 -8812.304,E2 -8812.304} C_VEL
LIN {X 0,Y 445.93,Z 578.305,A -85,B 0,C 180,E1 -8813.666,E2 -8813.666} C_VEL
LIN {X 0,Y 445.61,Z 582.394,A -85,B 0,C 180,E1 -8815.024,E2 -8815.024} C_VEL
LIN {X 0,Y 445.631,Z 585.376,A -85,B 0,C 180,E1 -8816.383,E2 -8816.383} C_VEL
LIN {X 0,Y 445.52,Z 586.818,A -85,B 0,C 180,E1 -8817.288,E2 -8817.288} C_VEL
LIN {X 0,Y 445.46,Z 587.805,A -85,B 0,C 180,E1 -8818.192,E2 -8818.192} C_VEL
LIN {X 0,Y 445.43,Z 588.393,A -85,B 0,C 180,E1 -8819.096,E2 -8819.096} C_VEL
LIN {X 0,Y 445.405,Z 588.57,A -85,B 0,C 180,E1 -8820,E2 -8820} C_VEL
LIN {X 0,Y 445.399,Z 588.29,A -85,B 0,C 180,E1 -8820.904,E2 -8820.904} C_VEL
LIN {X 0,Y 445.432,Z 587.607,A -85,B 0,C 180,E1 -8821.808,E2 -8821.808} C_VEL
LIN {X 0,Y 445.504,Z 586.522,A -85,B 0,C 180,E1 -8822.713,E2 -8822.713} C_VEL
LIN {X 0,Y 445.586,Z 584.971,A -85,B 0,C 180,E1 -8823.617,E2 -8823.617} C_VEL
LIN {X 0,Y 445.567,Z 581.826,A -85,B 0,C 180,E1 -8824.977,E2 -8824.977} C_VEL
LIN {X 0,Y 445.827,Z 577.578,A -85,B 0,C 180,E1 -8826.335,E2 -8826.335} C_VEL
LIN {X 0,Y 445.998,Z 571.104,A -85,B 0,C 180,E1 -8827.925,E2 -8827.925} C_VEL
LIN {X 0,Y 446.372,Z 563.968,A -85,B 0,C 180,E1 -8829.287,E2 -8829.287} C_VEL
LIN {X 0,Y 446.78,Z 555.072,A -85,B 0,C 180,E1 -8830.651,E2 -8830.651} C_VEL
LIN {X 0,Y 447.263,Z 545.925,A -85,B 0,C 180,E1 -8831.787,E2 -8831.787} C_VEL
LIN {X 0,Y 447.763,Z 535.406,A -85,B 0,C 180,E1 -8832.844,E2 -8832.844} C_VEL
LIN {X 0,Y 448.165,Z 524.644,A -85,B 0,C 180,E1 -8833.721,E2 -8833.721} C_VEL
LIN {X 0,Y 448.666,Z 512.091,A -85,B 0,C 180,E1 -8834.515,E2 -8834.515} C_VEL
LIN {X 0,Y 449.076,Z 498.827,A -85,B 0,C 180,E1 -8835.139,E2 -8835.139} C_VEL
LIN {X 0,Y 449.438,Z 485.365,A -85,B 0,C 180,E1 -8835.562,E2 -8835.562} C_VEL
LIN {X 0,Y 450.601,Z 391.687,A -85,B 0,C 180,E1 -8837.296,E2 -8837.296} C_VEL
LIN {X 0,Y 447.9,Z 376.31,A -85,B 0,C 180,E1 -8837.69,E2 -8837.69} C_VEL
LIN {X 0,Y 448.394,Z 358.223,A -85,B 0,C 180,E1 -8840.89,E2 -8840.89} C_VEL
